LIN {X 0,Y 207.025,Z 158.787,A -85,B 0,C 180,E1 -21118.588,E2 -21118.588} C_VEL
LIN {X 0,Y 213.281,Z 171.917,A -85,B 0,C 180,E1 -21120.162,E2 -21120.162} C_VEL
LIN {X 0,Y 219.22,Z 186.796,A -85,B 0,C 180,E1 -21121.599,E2 -21121.599} C_VEL
LIN {X 0,Y 220.481,Z 191.391,A -85,B 0,C 180,E1 -21121.944,E2 -21121.944} C_VEL
LIN {X 0,Y 221.304,Z 196.769,A -85,B 0,C 180,E1 -21122.252,E2 -21122.252} C_VEL
LIN {X 0,Y 219.851,Z 234.463,A -85,B 0,C 180,E1 -21123.468,E2 -21123.468} C_VEL
LIN {X 0,Y 219.142,Z 244.352,A -85,B 0,C 180,E1 -21124.024,E2 -21124.024} C_VEL
LIN {X 0,Y 218.068,Z 254.849,A -85,B 0,C 180,E1 -21124.912,E2 -21124.912} C_VEL
LIN {X 0,Y 216.311,Z 266.211,A -85,B 0,C 180,E1 -21126.292,E2 -21126.292} C_VEL
LIN {X 0,Y 214.803,Z 274.591,A -85,B 0,C 180,E1 -21127.644,E2 -21127.644} C_VEL
LIN {X 0,Y 213.065,Z 282.507,A -85,B 0,C 180,E1 -21129.231,E2 -21129.231} C_VEL
LIN {X 0,Y 211.348,Z 289.887,A -85,B 0,C 180,E1 -21131.081,E2 -21131.081} C_VEL
LIN {X 0,Y 209.44,Z 297.362,A -85,B 0,C 180,E1 -21133.427,E2 -21133.427} C_VEL
LIN {X 0,Y 207.589,Z 304.212,A -85,B 0,C 180,E1 -21136.291,E2 -21136.291} C_VEL
LIN {X 0,Y 206.206,Z 309.389,A -85,B 0,C 180,E1 -21139.195,E2 -21139.195} C_VEL
LIN {X 0,Y 205.508,Z 312.044,A -85,B 0,C 180,E1 -21141.147,E2 -21141.147} C_VEL
LIN {X 0,Y 204.74,Z 315.32,A -85,B 0,C 180,E1 -21144.544,E2 -21144.544} C_VEL
LIN {X 0,Y 204.386,Z 317.015,A -85,B 0,C 180,E1 -21148.029,E2 -21148.029} C_VEL
LIN {X 0,Y 204.39,Z 317.318,A -85,B 0,C 180,E1 -21150,E2 -21150} C_VEL
LIN {X 0,Y 204.385,Z 317.039,A -85,B 0,C 180,E1 -21151.97,E2 -21151.97} C_VEL
LIN {X 0,Y 204.716,Z 315.5,A -85,B 0,C 180,E1 -21155.384,E2 -21155.384} C_VEL
LIN {X 0,Y 205.209,Z 313.362,A -85,B 0,C 180,E1 -21157.873,E2 -21157.873} C_VEL
LIN {X 0,Y 206.179,Z 309.614,A -85,B 0,C 180,E1 -21160.805,E2 -21160.805} C_VEL
LIN {X 0,Y 207.558,Z 304.498,A -85,B 0,C 180,E1 -21163.71,E2 -21163.71} C_VEL
LIN {X 0,Y 209.032,Z 298.993,A -85,B 0,C 180,E1 -21166.103,E2 -21166.103} C_VEL
LIN {X 0,Y 210.882,Z 292.07,A -85,B 0,C 180,E1 -21168.457,E2 -21168.457} C_VEL
LIN {X 0,Y 212.763,Z 284.122,A -85,B 0,C 180,E1 -21170.546,E2 -21170.546} C_VEL
LIN {X 0,Y 214.475,Z 276.541,A -85,B 0,C 180,E1 -21172.137,E2 -21172.137} C_VEL
LIN {X 0,Y 216.015,Z 268.593,A -85,B 0,C 180,E1 -21173.487,E2 -21173.487} C_VEL
LIN {X 0,Y 217.416,Z 260.376,A -85,B 0,C 180,E1 -21174.593,E2 -21174.593} C_VEL
LIN {X 0,Y 218.618,Z 251.281,A -85,B 0,C 180,E1 -21175.545,E2 -21175.545} C_VEL
LIN {X 0,Y 219.566,Z 240.802,A -85,B 0,C 180,E1 -21176.344,E2 -21176.344} C_VEL
LIN {X 0,Y 220.274,Z 226.937,A -85,B 0,C 180,E1 -21176.954,E2 -21176.954} C_VEL
LIN {X 0,Y 221.254,Z 195.857,A -85,B 0,C 180,E1 -21177.938,E2 -21177.938} C_VEL
LIN {X 0,Y 219.854,Z 188.323,A -85,B 0,C 180,E1 -21178.407,E2 -21178.407} C_VEL
LIN {X 0,Y 213.607,Z 172.604,A -85,B 0,C 180,E1 -21179.917,E2 -21179.917} C_VEL
LIN {X 0,Y 208.077,Z 161.104,A -85,B 0,C 180,E1 -21181.255,E2 -21181.255} C_VEL
LIN {X 0,Y 206.898,Z 158.307,A -85,B 0,C 180,E1 -21181.691,E2 -21181.691} C_VEL
LIN {X 0,Y 206.732,Z 157.678,A -85,B 0,C 180,E1 -21182.04,E2 -21182.04} C_VEL
LIN {X 0,Y 206.722,Z 157.517,A -85,B 0,C 180,E1 -21185.32,E2 -21185.32} C_VEL
LIN {X 0,Y 206.665,Z 157.531,A -85,B 0,C 180,E1 -21190.25,E2 -21190.25} C_VEL
LIN {X 0,Y 206.631,Z 157.549,A -85,B 0,C 180,E1 -21195.582,E2 -21195.582} C_VEL
LIN {X 0,Y 206.66,Z 157.542,A -85,B 0,C 180,E1 -21199.748,E2 -21199.748} C_VEL
LIN {X 0,Y 206.698,Z 157.542,A -85,B 0,C 180,E1 -21204.688,E2 -21204.688} C_VEL
LIN {X 0,Y 206.723,Z 157.548,A -85,B 0,C 180,E1 -21209.339,E2 -21209.339} C_VEL
LIN {X 0,Y 206.731,Z 157.525,A -85,B 0,C 180,E1 -21213.772,E2 -21213.772} C_VEL
LIN {X 0,Y 206.757,Z 157.542,A -85,B 0,C 180,E1 -21218.043,E2 -21218.043} C_VEL
LIN {X 0,Y 206.872,Z 157.503,A -85,B 0,C 180,E1 -21222.196,E2 -21222.196} C_VEL
LIN {X 0,Y 206.914,Z 157.523,A -85,B 0,C 180,E1 -21226.245,E2 -21226.245} C_VEL
LIN {X 0,Y 207.105,Z 157.474,A -85,B 0,C 180,E1 -21230.231,E2 -21230.231} C_VEL
LIN {X 0,Y 207.167,Z 157.468,A -85,B 0,C 180,E1 -21232.201,E2 -21232.201} C_VEL
LIN {X 0,Y 207.382,Z 157.456,A -85,B 0,C 180,E1 -21238.058,E2 -21238.058} C_VEL
LIN {X 0,Y 207.514,Z 157.421,A -85,B 0,C 180,E1 -21240,E2 -21240} C_VEL
LIN {X 0,Y 207.382,Z 157.44,A -85,B 0,C 180,E1 -21241.942,E2 -21241.942} C_VEL
LIN {X 0,Y 207.178,Z 157.481,A -85,B 0,C 180,E1 -21247.798,E2 -21247.798} C_VEL
LIN {X 0,Y 206.98,Z 157.493,A -85,B 0,C 180,E1 -21251.755,E2 -21251.755} C_VEL
LIN {X 0,Y 206.866,Z 157.528,A -85,B 0,C 180,E1 -21255.771,E2 -21255.771} C_VEL
LIN {X 0,Y 206.782,Z 157.516,A -85,B 0,C 180,E1 -21259.869,E2 -21259.869} C_VEL
LIN {X 0,Y 206.762,Z 157.542,A -85,B 0,C 180,E1 -21264.072,E2 -21264.072} C_VEL
LIN {X 0,Y 206.743,Z 157.526,A -85,B 0,C 180,E1 -21268.419,E2 -21268.419} C_VEL
LIN {X 0,Y 206.701,Z 157.544,A -85,B 0,C 180,E1 -21272.957,E2 -21272.957} C_VEL
LIN {X 0,Y 206.679,Z 157.553,A -85,B 0,C 180,E1 -21277.74,E2 -21277.74} C_VEL
LIN {X 0,Y 206.639,Z 157.518,A -85,B 0,C 180,E1 -21281.562,E2 -21281.562} C_VEL
LIN {X 0,Y 206.629,Z 157.526,A -85,B 0,C 180,E1 -21285.583,E2 -21285.583} C_VEL
LIN {X 0,Y 206.658,Z 157.54,A -85,B 0,C 180,E1 -21289.749,E2 -21289.749} C_VEL
LIN {X 0,Y 206.714,Z 157.652,A -85,B 0,C 180,E1 -21294.558,E2 -21294.558} C_VEL
LIN {X 0,Y 208.276,Z 164.486,A -85,B 0,C 180,E1 -21298.581,E2 -21298.581} C_VEL
LIN {X 0,Y 209.79,Z 168.116,A -85,B 0,C 180,E1 -21299.094,E2 -21299.094} C_VEL
LIN {X 0,Y 213.712,Z 177.001,A -85,B 0,C 180,E1 -21300.057,E2 -21300.057} C_VEL
LIN {X 0,Y 214.926,Z 182.58,A -85,B 0,C 180,E1 -21300.452,E2 -21300.452} C_VEL
LIN {X 0,Y 215.138,Z 188.446,A -85,B 0,C 180,E1 -21300.704,E2 -21300.704} C_VEL
LIN {X 0,Y 214.129,Z 204.462,A -85,B 0,C 180,E1 -21301.155,E2 -21301.155} C_VEL
LIN {X 0,Y 214.248,Z 208.452,A -85,B 0,C 180,E1 -21301.322,E2 -21301.322} C_VEL
LIN {X 0,Y 214.544,Z 211.919,A -85,B 0,C 180,E1 -21301.494,E2 -21301.494} C_VEL
LIN {X 0,Y 213.364,Z 242.504,A -85,B 0,C 180,E1 -21302.539,E2 -21302.539} C_VEL
LIN {X 0,Y 212.457,Z 252.749,A -85,B 0,C 180,E1 -21303.145,E2 -21303.145} C_VEL
LIN {X 0,Y 211.077,Z 263.496,A -85,B 0,C 180,E1 -21304.114,E2 -21304.114} C_VEL
LIN {X 0,Y 209.3,Z 273.86,A -85,B 0,C 180,E1 -21305.448,E2 -21305.448} C_VEL
LIN {X 0,Y 207.628,Z 282.146,A -85,B 0,C 180,E1 -21306.828,E2 -21306.828} C_VEL
LIN {X 0,Y 205.824,Z 289.992,A -85,B 0,C 180,E1 -21308.466,E2 -21308.466} C_VEL
LIN {X 0,Y 203.943,Z 297.33,A -85,B 0,C 180,E1 -21310.368,E2 -21310.368} C_VEL
LIN {X 0,Y 201.943,Z 304.775,A -85,B 0,C 180,E1 -21312.794,E2 -21312.794} C_VEL
LIN {X 0,Y 200.353,Z 310.611,A -85,B 0,C 180,E1 -21315.267,E2 -21315.267} C_VEL
LIN {X 0,Y 199.065,Z 315.214,A -85,B 0,C 180,E1 -21317.771,E2 -21317.771} C_VEL
LIN {X 0,Y 198.362,Z 318.207,A -85,B 0,C 180,E1 -21319.797,E2 -21319.797} C_VEL
LIN {X 0,Y 197.78,Z 320.53,A -85,B 0,C 180,E1 -21321.829,E2 -21321.829} C_VEL
LIN {X 0,Y 197.427,Z 322.272,A -85,B 0,C 180,E1 -21323.87,E2 -21323.87} C_VEL
LIN {X 0,Y 197.237,Z 323.613,A -85,B 0,C 180,E1 -21326.113,E2 -21326.113} C_VEL
LIN {X 0,Y 197.214,Z 324.293,A -85,B 0,C 180,E1 -21327.958,E2 -21327.958} C_VEL
LIN {X 0,Y 197.252,Z 324.585,A -85,B 0,C 180,E1 -21330,E2 -21330} C_VEL
LIN {X 0,Y 197.214,Z 324.283,A -85,B 0,C 180,E1 -21332.043,E2 -21332.043} C_VEL
LIN {X 0,Y 197.25,Z 323.49,A -85,B 0,C 180,E1 -21334.087,E2 -21334.087} C_VEL
LIN {X 0,Y 197.43,Z 322.223,A -85,B 0,C 180,E1 -21336.131,E2 -21336.131} C_VEL
LIN {X 0,Y 198.004,Z 319.305,A -85,B 0,C 180,E1 -21339.191,E2 -21339.191} C_VEL
LIN {X 0,Y 198.649,Z 316.646,A -85,B 0,C 180,E1 -21341.221,E2 -21341.221} C_VEL
LIN {X 0,Y 200.061,Z 311.454,A -85,B 0,C 180,E1 -21344.236,E2 -21344.236} C_VEL
LIN {X 0,Y 201.922,Z 304.606,A -85,B 0,C 180,E1 -21347.209,E2 -21347.209} C_VEL
LIN {X 0,Y 203.932,Z 297.128,A -85,B 0,C 180,E1 -21349.634,E2 -21349.634} C_VEL
LIN {X 0,Y 205.828,Z 289.754,A -85,B 0,C 180,E1 -21351.535,E2 -21351.535} C_VEL
LIN {X 0,Y 207.584,Z 281.852,A -85,B 0,C 180,E1 -21353.178,E2 -21353.178} C_VEL
LIN {X 0,Y 209.567,Z 272.214,A -85,B 0,C 180,E1 -21354.746,E2 -21354.746} C_VEL
LIN {X 0,Y 211.277,Z 261.067,A -85,B 0,C 180,E1 -21356.086,E2 -21356.086} C_VEL
LIN {X 0,Y 212.53,Z 251.125,A -85,B 0,C 180,E1 -21356.912,E2 -21356.912} C_VEL
LIN {X 0,Y 213.384,Z 241.25,A -85,B 0,C 180,E1 -21357.459,E2 -21357.459} C_VEL
LIN {X 0,Y 214.439,Z 210.557,A -85,B 0,C 180,E1 -21358.508,E2 -21358.508} C_VEL
LIN {X 0,Y 211.33,Z 188.673,A -85,B 0,C 180,E1 -21359.799,E2 -21359.799} C_VEL
LIN {X 0,Y 205.481,Z 174.284,A -85,B 0,C 180,E1 -21361.306,E2 -21361.306} C_VEL
LIN {X 0,Y 201.105,Z 164.731,A -85,B 0,C 180,E1 -21362.512,E2 -21362.512} C_VEL
LIN {X 0,Y 200.705,Z 163.01,A -85,B 0,C 180,E1 -21363.337,E2 -21363.337} C_VEL
LIN {X 0,Y 199.673,Z 158.489,A -85,B 0,C 180,E1 -21366.258,E2 -21366.258} C_VEL
LIN {X 0,Y 199.608,Z 158.407,A -85,B 0,C 180,E1 -21369.329,E2 -21369.329} C_VEL
LIN {X 0,Y 199.573,Z 158.437,A -85,B 0,C 180,E1 -21372.31,E2 -21372.31} C_VEL
LIN {X 0,Y 199.577,Z 158.389,A -85,B 0,C 180,E1 -21375.228,E2 -21375.228} C_VEL
LIN {X 0,Y 199.578,Z 158.39,A -85,B 0,C 180,E1 -21378.005,E2 -21378.005} C_VEL
LIN {X 0,Y 199.612,Z 158.43,A -85,B 0,C 180,E1 -21380.768,E2 -21380.768} C_VEL
LIN {X 0,Y 199.614,Z 158.418,A -85,B 0,C 180,E1 -21385.714,E2 -21385.714} C_VEL
LIN {X 0,Y 199.702,Z 158.422,A -85,B 0,C 180,E1 -21388.138,E2 -21388.138} C_VEL
LIN {X 0,Y 199.688,Z 158.402,A -85,B 0,C 180,E1 -21392.772,E2 -21392.772} C_VEL
LIN {X 0,Y 199.74,Z 158.414,A -85,B 0,C 180,E1 -21397.23,E2 -21397.23} C_VEL
LIN {X 0,Y 199.799,Z 158.392,A -85,B 0,C 180,E1 -21401.758,E2 -21401.758} C_VEL
LIN {X 0,Y 199.838,Z 158.403,A -85,B 0,C 180,E1 -21405.749,E2 -21405.749} C_VEL
LIN {X 0,Y 200.024,Z 158.352,A -85,B 0,C 180,E1 -21409.882,E2 -21409.882} C_VEL
LIN {X 0,Y 200.029,Z 158.38,A -85,B 0,C 180,E1 -21413.95,E2 -21413.95} C_VEL
LIN {X 0,Y 200.323,Z 158.318,A -85,B 0,C 180,E1 -21417.99,E2 -21417.99} C_VEL
LIN {X 0,Y 200.479,Z 158.296,A -85,B 0,C 180,E1 -21420,E2 -21420} C_VEL
LIN {X 0,Y 200.034,Z 158.382,A -85,B 0,C 180,E1 -21424.03,E2 -21424.03} C_VEL
LIN {X 0,Y 200.114,Z 158.343,A -85,B 0,C 180,E1 -21428.076,E2 -21428.076} C_VEL
LIN {X 0,Y 199.917,Z 158.39,A -85,B 0,C 180,E1 -21432.177,E2 -21432.177} C_VEL
LIN {X 0,Y 199.807,Z 158.395,A -85,B 0,C 180,E1 -21436.343,E2 -21436.343} C_VEL
LIN {X 0,Y 199.703,Z 158.413,A -85,B 0,C 180,E1 -21440.605,E2 -21440.605} C_VEL
LIN {X 0,Y 199.675,Z 158.411,A -85,B 0,C 180,E1 -21444.984,E2 -21444.984} C_VEL
LIN {X 0,Y 199.677,Z 158.424,A -85,B 0,C 180,E1 -21449.522,E2 -21449.522} C_VEL
LIN {X 0,Y 199.68,Z 158.414,A -85,B 0,C 180,E1 -21452.358,E2 -21452.358} C_VEL
LIN {X 0,Y 199.625,Z 158.432,A -85,B 0,C 180,E1 -21456.763,E2 -21456.763} C_VEL
LIN {X 0,Y 199.61,Z 158.422,A -85,B 0,C 180,E1 -21459.328,E2 -21459.328} C_VEL
LIN {X 0,Y 199.576,Z 158.438,A -85,B 0,C 180,E1 -21462.31,E2 -21462.31} C_VEL
LIN {X 0,Y 199.579,Z 158.413,A -85,B 0,C 180,E1 -21465.228,E2 -21465.228} C_VEL
LIN {X 0,Y 199.641,Z 158.419,A -85,B 0,C 180,E1 -21470.679,E2 -21470.679} C_VEL
LIN {X 0,Y 199.636,Z 158.399,A -85,B 0,C 180,E1 -21475.718,E2 -21475.718} C_VEL
LIN {X 0,Y 199.714,Z 158.737,A -85,B 0,C 180,E1 -21477.093,E2 -21477.093} C_VEL
LIN {X 0,Y 200.101,Z 160.119,A -85,B 0,C 180,E1 -21477.452,E2 -21477.452} C_VEL
LIN {X 0,Y 203.509,Z 166.286,A -85,B 0,C 180,E1 -21478.333,E2 -21478.333} C_VEL
LIN {X 0,Y 210.222,Z 181.264,A -85,B 0,C 180,E1 -21480.042,E2 -21480.042} C_VEL
LIN {X 0,Y 214.246,Z 192.387,A -85,B 0,C 180,E1 -21481.083,E2 -21481.083} C_VEL
LIN {X 0,Y 215.01,Z 197.207,A -85,B 0,C 180,E1 -21481.376,E2 -21481.376} C_VEL
LIN {X 0,Y 213.523,Z 234.798,A -85,B 0,C 180,E1 -21482.626,E2 -21482.626} C_VEL
LIN {X 0,Y 212.788,Z 244.531,A -85,B 0,C 180,E1 -21483.19,E2 -21483.19} C_VEL
LIN {X 0,Y 211.656,Z 255.205,A -85,B 0,C 180,E1 -21484.121,E2 -21484.121} C_VEL
LIN {X 0,Y 209.848,Z 266.344,A -85,B 0,C 180,E1 -21485.515,E2 -21485.515} C_VEL
LIN {X 0,Y 208.27,Z 274.723,A -85,B 0,C 180,E1 -21486.903,E2 -21486.903} C_VEL
LIN {X 0,Y 206.459,Z 282.638,A -85,B 0,C 180,E1 -21488.534,E2 -21488.534} C_VEL
LIN {X 0,Y 205.046,Z 288.32,A -85,B 0,C 180,E1 -21489.955,E2 -21489.955} C_VEL
LIN {X 0,Y 203.393,Z 294.666,A -85,B 0,C 180,E1 -21491.881,E2 -21491.881} C_VEL
LIN {X 0,Y 201.929,Z 299.94,A -85,B 0,C 180,E1 -21493.833,E2 -21493.833} C_VEL
LIN {X 0,Y 200.693,Z 304.342,A -85,B 0,C 180,E1 -21495.81,E2 -21495.81} C_VEL
LIN {X 0,Y 199.23,Z 309.519,A -85,B 0,C 180,E1 -21498.812,E2 -21498.812} C_VEL
LIN {X 0,Y 198.486,Z 312.173,A -85,B 0,C 180,E1 -21500.831,E2 -21500.831} C_VEL
LIN {X 0,Y 197.767,Z 315.079,A -85,B 0,C 180,E1 -21503.88,E2 -21503.88} C_VEL
LIN {X 0,Y 197.467,Z 316.345,A -85,B 0,C 180,E1 -21505.918,E2 -21505.918} C_VEL
LIN {X 0,Y 197.299,Z 317.143,A -85,B 0,C 180,E1 -21507.958,E2 -21507.958} C_VEL
LIN {X 0,Y 197.296,Z 317.446,A -85,B 0,C 180,E1 -21510,E2 -21510} C_VEL
LIN {X 0,Y 197.298,Z 317.167,A -85,B 0,C 180,E1 -21512.041,E2 -21512.041} C_VEL
LIN {X 0,Y 197.6,Z 315.877,A -85,B 0,C 180,E1 -21515.205,E2 -21515.205} C_VEL
LIN {X 0,Y 198.175,Z 313.49,A -85,B 0,C 180,E1 -21518.155,E2 -21518.155} C_VEL
LIN {X 0,Y 199.204,Z 309.741,A -85,B 0,C 180,E1 -21521.188,E2 -21521.188} C_VEL
LIN {X 0,Y 200.657,Z 304.625,A -85,B 0,C 180,E1 -21524.192,E2 -21524.192} C_VEL
LIN {X 0,Y 202.219,Z 299.119,A -85,B 0,C 180,E1 -21526.661,E2 -21526.661} C_VEL
LIN {X 0,Y 204.159,Z 292.196,A -85,B 0,C 180,E1 -21529.088,E2 -21529.088} C_VEL
LIN {X 0,Y 206.148,Z 284.247,A -85,B 0,C 180,E1 -21531.237,E2 -21531.237} C_VEL
LIN {X 0,Y 207.937,Z 276.665,A -85,B 0,C 180,E1 -21532.872,E2 -21532.872} C_VEL
LIN {X 0,Y 209.542,Z 268.716,A -85,B 0,C 180,E1 -21534.258,E2 -21534.258} C_VEL
LIN {X 0,Y 210.987,Z 260.498,A -85,B 0,C 180,E1 -21535.395,E2 -21535.395} C_VEL
LIN {X 0,Y 212.159,Z 252.232,A -85,B 0,C 180,E1 -21536.291,E2 -21536.291} C_VEL
LIN {X 0,Y 213.083,Z 242.81,A -85,B 0,C 180,E1 -21537.06,E2 -21537.06} C_VEL
LIN {X 0,Y 213.691,Z 233.428,A -85,B 0,C 180,E1 -21537.574,E2 -21537.574} C_VEL
LIN {X 0,Y 215.027,Z 197.05,A -85,B 0,C 180,E1 -21538.781,E2 -21538.781} C_VEL
LIN {X 0,Y 213.929,Z 191.058,A -85,B 0,C 180,E1 -21539.169,E2 -21539.169} C_VEL
LIN {X 0,Y 208.339,Z 176.751,A -85,B 0,C 180,E1 -21540.595,E2 -21540.595} C_VEL
LIN {X 0,Y 202.889,Z 165.209,A -85,B 0,C 180,E1 -21541.984,E2 -21541.984} C_VEL
LIN {X 0,Y 200.65,Z 161.212,A -85,B 0,C 180,E1 -21542.552,E2 -21542.552} C_VEL
LIN {X 0,Y 199.794,Z 159.117,A -85,B 0,C 180,E1 -21542.912,E2 -21542.912} C_VEL
LIN {X 0,Y 199.67,Z 158.533,A -85,B 0,C 180,E1 -21543.244,E2 -21543.244} C_VEL
LIN {X 0,Y 199.619,Z 158.41,A -85,B 0,C 180,E1 -21546.763,E2 -21546.763} C_VEL
LIN {X 0,Y 199.639,Z 158.424,A -85,B 0,C 180,E1 -21549.32,E2 -21549.32} C_VEL
LIN {X 0,Y 199.577,Z 158.409,A -85,B 0,C 180,E1 -21554.771,E2 -21554.771} C_VEL
LIN {X 0,Y 199.578,Z 158.437,A -85,B 0,C 180,E1 -21558.004,E2 -21558.004} C_VEL
LIN {X 0,Y 199.61,Z 158.421,A -85,B 0,C 180,E1 -21560.767,E2 -21560.767} C_VEL
LIN {X 0,Y 199.612,Z 158.415,A -85,B 0,C 180,E1 -21565.713,E2 -21565.713} C_VEL
LIN {X 0,Y 199.7,Z 158.416,A -85,B 0,C 180,E1 -21568.137,E2 -21568.137} C_VEL
LIN {X 0,Y 199.686,Z 158.404,A -85,B 0,C 180,E1 -21572.771,E2 -21572.771} C_VEL
LIN {X 0,Y 199.738,Z 158.417,A -85,B 0,C 180,E1 -21577.229,E2 -21577.229} C_VEL
LIN {X 0,Y 199.796,Z 158.383,A -85,B 0,C 180,E1 -21581.757,E2 -21581.757} C_VEL
LIN {X 0,Y 199.848,Z 158.402,A -85,B 0,C 180,E1 -21585.749,E2 -21585.749} C_VEL
LIN {X 0,Y 200.069,Z 158.352,A -85,B 0,C 180,E1 -21589.884,E2 -21589.884} C_VEL
LIN {X 0,Y 200.035,Z 158.372,A -85,B 0,C 180,E1 -21593.949,E2 -21593.949} C_VEL
LIN {X 0,Y 200.322,Z 158.335,A -85,B 0,C 180,E1 -21597.989,E2 -21597.989} C_VEL
LIN {X 0,Y 200.479,Z 158.297,A -85,B 0,C 180,E1 -21600,E2 -21600} C_VEL
LIN {X 0,Y 200.031,Z 158.374,A -85,B 0,C 180,E1 -21604.029,E2 -21604.029} C_VEL
LIN {X 0,Y 200.119,Z 158.359,A -85,B 0,C 180,E1 -21608.075,E2 -21608.075} C_VEL
LIN {X 0,Y 199.913,Z 158.377,A -85,B 0,C 180,E1 -21612.177,E2 -21612.177} C_VEL
LIN {X 0,Y 199.804,Z 158.406,A -85,B 0,C 180,E1 -21616.343,E2 -21616.343} C_VEL
LIN {X 0,Y 199.699,Z 158.401,A -85,B 0,C 180,E1 -21620.605,E2 -21620.605} C_VEL
LIN {X 0,Y 199.672,Z 158.422,A -85,B 0,C 180,E1 -21624.984,E2 -21624.984} C_VEL
LIN {X 0,Y 199.673,Z 158.415,A -85,B 0,C 180,E1 -21629.522,E2 -21629.522} C_VEL
LIN {X 0,Y 199.676,Z 158.423,A -85,B 0,C 180,E1 -21632.358,E2 -21632.358} C_VEL
LIN {X 0,Y 199.622,Z 158.428,A -85,B 0,C 180,E1 -21636.763,E2 -21636.763} C_VEL
LIN {X 0,Y 199.607,Z 158.428,A -85,B 0,C 180,E1 -21639.328,E2 -21639.328} C_VEL
LIN {X 0,Y 199.57,Z 158.388,A -85,B 0,C 180,E1 -21642.31,E2 -21642.31} C_VEL
LIN {X 0,Y 199.575,Z 158.396,A -85,B 0,C 180,E1 -21645.228,E2 -21645.228} C_VEL
LIN {X 0,Y 199.577,Z 158.439,A -85,B 0,C 180,E1 -21648.005,E2 -21648.005} C_VEL
LIN {X 0,Y 199.653,Z 158.405,A -85,B 0,C 180,E1 -21653.244,E2 -21653.244} C_VEL
LIN {X 0,Y 199.727,Z 158.927,A -85,B 0,C 180,E1 -21654.03,E2 -21654.03} C_VEL
LIN {X 0,Y 201.015,Z 164.444,A -85,B 0,C 180,E1 -21657.335,E2 -21657.335} C_VEL
LIN {X 0,Y 203.312,Z 169.666,A -85,B 0,C 180,E1 -21658.063,E2 -21658.063} C_VEL
LIN {X 0,Y 208.434,Z 181.104,A -85,B 0,C 180,E1 -21659.382,E2 -21659.382} C_VEL
LIN {X 0,Y 211.571,Z 189.597,A -85,B 0,C 180,E1 -21660.207,E2 -21660.207} C_VEL
LIN {X 0,Y 214.248,Z 208.452,A -85,B 0,C 180,E1 -21661.322,E2 -21661.322} C_VEL
LIN {X 0,Y 214.19,Z 212.339,A -85,B 0,C 180,E1 -21661.454,E2 -21661.454} C_VEL
LIN {X 0,Y 213.558,Z 216.217,A -85,B 0,C 180,E1 -21661.496,E2 -21661.496} C_VEL
LIN {X 0,Y 208.229,Z 233.389,A -85,B 0,C 180,E1 -21661.352,E2 -21661.352} C_VEL
LIN {X 0,Y 207.287,Z 239.256,A -85,B 0,C 180,E1 -21661.496,E2 -21661.496} C_VEL
LIN {X 0,Y 206.51,Z 249.311,A -85,B 0,C 180,E1 -21662.031,E2 -21662.031} C_VEL
LIN {X 0,Y 205.36,Z 258.749,A -85,B 0,C 180,E1 -21662.788,E2 -21662.788} C_VEL
LIN {X 0,Y 203.979,Z 267.807,A -85,B 0,C 180,E1 -21663.794,E2 -21663.794} C_VEL
LIN {X 0,Y 202.24,Z 276.884,A -85,B 0,C 180,E1 -21665.107,E2 -21665.107} C_VEL
LIN {X 0,Y 200.02,Z 286.799,A -85,B 0,C 180,E1 -21666.991,E2 -21666.991} C_VEL
LIN {X 0,Y 197.726,Z 295.497,A -85,B 0,C 180,E1 -21669.18,E2 -21669.18} C_VEL
LIN {X 0,Y 195.949,Z 301.815,A -85,B 0,C 180,E1 -21671.168,E2 -21671.168} C_VEL
LIN {X 0,Y 194.402,Z 307.064,A -85,B 0,C 180,E1 -21673.19,E2 -21673.19} C_VEL
LIN {X 0,Y 193.175,Z 311.443,A -85,B 0,C 180,E1 -21675.246,E2 -21675.246} C_VEL
LIN {X 0,Y 191.716,Z 316.609,A -85,B 0,C 180,E1 -21678.369,E2 -21678.369} C_VEL
LIN {X 0,Y 190.748,Z 320.403,A -85,B 0,C 180,E1 -21681.526,E2 -21681.526} C_VEL
LIN {X 0,Y 190.369,Z 322.144,A -85,B 0,C 180,E1 -21683.642,E2 -21683.642} C_VEL
LIN {X 0,Y 190.142,Z 323.657,A -85,B 0,C 180,E1 -21686.344,E2 -21686.344} C_VEL
LIN {X 0,Y 190.161,Z 324.457,A -85,B 0,C 180,E1 -21690.001,E2 -21690.001} C_VEL
LIN {X 0,Y 190.142,Z 323.627,A -85,B 0,C 180,E1 -21693.657,E2 -21693.657} C_VEL
LIN {X 0,Y 190.372,Z 322.094,A -85,B 0,C 180,E1 -21696.359,E2 -21696.359} C_VEL
LIN {X 0,Y 190.998,Z 319.176,A -85,B 0,C 180,E1 -21699.532,E2 -21699.532} C_VEL
LIN {X 0,Y 191.685,Z 316.516,A -85,B 0,C 180,E1 -21701.634,E2 -21701.634} C_VEL
LIN {X 0,Y 193.172,Z 311.323,A -85,B 0,C 180,E1 -21704.755,E2 -21704.755} C_VEL
LIN {X 0,Y 195.145,Z 304.475,A -85,B 0,C 180,E1 -21707.826,E2 -21707.826} C_VEL
LIN {X 0,Y 197.251,Z 296.997,A -85,B 0,C 180,E1 -21710.328,E2 -21710.328} C_VEL
LIN {X 0,Y 199.232,Z 289.622,A -85,B 0,C 180,E1 -21712.285,E2 -21712.285} C_VEL
LIN {X 0,Y 201.076,Z 281.72,A -85,B 0,C 180,E1 -21713.974,E2 -21713.974} C_VEL
LIN {X 0,Y 203.062,Z 272.531,A -85,B 0,C 180,E1 -21715.513,E2 -21715.513} C_VEL
LIN {X 0,Y 204.763,Z 262.276,A -85,B 0,C 180,E1 -21716.825,E2 -21716.825} C_VEL
LIN {X 0,Y 206.229,Z 250.986,A -85,B 0,C 180,E1 -21717.804,E2 -21717.804} C_VEL
LIN {X 0,Y 207.114,Z 241.105,A -85,B 0,C 180,E1 -21718.364,E2 -21718.364} C_VEL
LIN {X 0,Y 208.201,Z 211.301,A -85,B 0,C 180,E1 -21719.41,E2 -21719.41} C_VEL
LIN {X 0,Y 205.304,Z 190.857,A -85,B 0,C 180,E1 -21720.674,E2 -21720.674} C_VEL
LIN {X 0,Y 199.891,Z 177.49,A -85,B 0,C 180,E1 -21722.146,E2 -21722.146} C_VEL
LIN {X 0,Y 193.873,Z 164.661,A -85,B 0,C 180,E1 -21723.873,E2 -21723.873} C_VEL
LIN {X 0,Y 193.55,Z 163.504,A -85,B 0,C 180,E1 -21724.374,E2 -21724.374} C_VEL
LIN {X 0,Y 192.605,Z 159.381,A -85,B 0,C 180,E1 -21727.149,E2 -21727.149} C_VEL
LIN {X 0,Y 192.513,Z 159.313,A -85,B 0,C 180,E1 -21731.081,E2 -21731.081} C_VEL
LIN {X 0,Y 192.489,Z 159.264,A -85,B 0,C 180,E1 -21736.076,E2 -21736.076} C_VEL
LIN {X 0,Y 192.519,Z 159.303,A -85,B 0,C 180,E1 -21740.052,E2 -21740.052} C_VEL
LIN {X 0,Y 192.562,Z 159.297,A -85,B 0,C 180,E1 -21744.271,E2 -21744.271} C_VEL
LIN {X 0,Y 192.612,Z 159.299,A -85,B 0,C 180,E1 -21747.059,E2 -21747.059} C_VEL
LIN {X 0,Y 192.666,Z 159.276,A -85,B 0,C 180,E1 -21751.692,E2 -21751.692} C_VEL
LIN {X 0,Y 192.708,Z 159.293,A -85,B 0,C 180,E1 -21756.349,E2 -21756.349} C_VEL
LIN {X 0,Y 192.734,Z 159.268,A -85,B 0,C 180,E1 -21761.458,E2 -21761.458} C_VEL
LIN {X 0,Y 192.766,Z 159.285,A -85,B 0,C 180,E1 -21765.214,E2 -21765.214} C_VEL
LIN {X 0,Y 192.947,Z 159.232,A -85,B 0,C 180,E1 -21769.567,E2 -21769.567} C_VEL
LIN {X 0,Y 193.044,Z 159.236,A -85,B 0,C 180,E1 -21771.627,E2 -21771.627} C_VEL
LIN {X 0,Y 193.265,Z 159.197,A -85,B 0,C 180,E1 -21777.916,E2 -21777.916} C_VEL
LIN {X 0,Y 193.443,Z 159.171,A -85,B 0,C 180,E1 -21780,E2 -21780} C_VEL
LIN {X 0,Y 192.98,Z 159.259,A -85,B 0,C 180,E1 -21784.177,E2 -21784.177} C_VEL
LIN {X 0,Y 193.065,Z 159.219,A -85,B 0,C 180,E1 -21788.373,E2 -21788.373} C_VEL
LIN {X 0,Y 192.856,Z 159.272,A -85,B 0,C 180,E1 -21792.63,E2 -21792.63} C_VEL
LIN {X 0,Y 192.76,Z 159.264,A -85,B 0,C 180,E1 -21796.959,E2 -21796.959} C_VEL
LIN {X 0,Y 192.639,Z 159.297,A -85,B 0,C 180,E1 -21801.397,E2 -21801.397} C_VEL
LIN {X 0,Y 192.667,Z 159.291,A -85,B 0,C 180,E1 -21804.225,E2 -21804.225} C_VEL
LIN {X 0,Y 192.652,Z 159.293,A -85,B 0,C 180,E1 -21808.892,E2 -21808.892} C_VEL
LIN {X 0,Y 192.601,Z 159.288,A -85,B 0,C 180,E1 -21813.186,E2 -21813.186} C_VEL
LIN {X 0,Y 192.553,Z 159.307,A -85,B 0,C 180,E1 -21818.352,E2 -21818.352} C_VEL
LIN {X 0,Y 192.513,Z 159.319,A -85,B 0,C 180,E1 -21823.102,E2 -21823.102} C_VEL
LIN {X 0,Y 192.492,Z 159.275,A -85,B 0,C 180,E1 -21826.905,E2 -21826.905} C_VEL
LIN {X 0,Y 192.57,Z 159.312,A -85,B 0,C 180,E1 -21831.652,E2 -21831.652} C_VEL
LIN {X 0,Y 192.634,Z 159.466,A -85,B 0,C 180,E1 -21835.652,E2 -21835.652} C_VEL
LIN {X 0,Y 192.845,Z 160.453,A -85,B 0,C 180,E1 -21836.058,E2 -21836.058} C_VEL
LIN {X 0,Y 198.456,Z 170.644,A -85,B 0,C 180,E1 -21837.607,E2 -21837.607} C_VEL
LIN {X 0,Y 204.768,Z 184.91,A -85,B 0,C 180,E1 -21839.299,E2 -21839.299} C_VEL
LIN {X 0,Y 208.232,Z 194.678,A -85,B 0,C 180,E1 -21840.249,E2 -21840.249} C_VEL
LIN {X 0,Y 208.808,Z 198.406,A -85,B 0,C 180,E1 -21840.484,E2 -21840.484} C_VEL
LIN {X 0,Y 207.242,Z 235.122,A -85,B 0,C 180,E1 -21841.733,E2 -21841.733} C_VEL
LIN {X 0,Y 206.455,Z 245.188,A -85,B 0,C 180,E1 -21842.341,E2 -21842.341} C_VEL
LIN {X 0,Y 205.12,Z 256.721,A -85,B 0,C 180,E1 -21843.411,E2 -21843.411} C_VEL
LIN {X 0,Y 203.428,Z 266.477,A -85,B 0,C 180,E1 -21844.689,E2 -21844.689} C_VEL
LIN {X 0,Y 201.778,Z 274.856,A -85,B 0,C 180,E1 -21846.114,E2 -21846.114} C_VEL
LIN {X 0,Y 199.877,Z 282.77,A -85,B 0,C 180,E1 -21847.791,E2 -21847.791} C_VEL
LIN {X 0,Y 198.404,Z 288.451,A -85,B 0,C 180,E1 -21849.253,E2 -21849.253} C_VEL
LIN {X 0,Y 196.655,Z 294.797,A -85,B 0,C 180,E1 -21851.237,E2 -21851.237} C_VEL
LIN {X 0,Y 195.126,Z 300.07,A -85,B 0,C 180,E1 -21853.253,E2 -21853.253} C_VEL
LIN {X 0,Y 193.8,Z 304.472,A -85,B 0,C 180,E1 -21855.294,E2 -21855.294} C_VEL
LIN {X 0,Y 192.277,Z 309.648,A -85,B 0,C 180,E1 -21858.402,E2 -21858.402} C_VEL
LIN {X 0,Y 191.486,Z 312.303,A -85,B 0,C 180,E1 -21860.493,E2 -21860.493} C_VEL
LIN {X 0,Y 190.725,Z 315.207,A -85,B 0,C 180,E1 -21863.653,E2 -21863.653} C_VEL
LIN {X 0,Y 190.405,Z 316.474,A -85,B 0,C 180,E1 -21865.766,E2 -21865.766} C_VEL
LIN {X 0,Y 190.214,Z 317.272,A -85,B 0,C 180,E1 -21867.882,E2 -21867.882} C_VEL
LIN {X 0,Y 190.204,Z 317.574,A -85,B 0,C 180,E1 -21869.999,E2 -21869.999} C_VEL
LIN {X 0,Y 190.213,Z 317.295,A -85,B 0,C 180,E1 -21872.117,E2 -21872.117} C_VEL
LIN {X 0,Y 190.497,Z 316.174,A -85,B 0,C 180,E1 -21875.052,E2 -21875.052} C_VEL
LIN {X 0,Y 191.14,Z 313.617,A -85,B 0,C 180,E1 -21878.457,E2 -21878.457} C_VEL
LIN {X 0,Y 192.249,Z 309.869,A -85,B 0,C 180,E1 -21881.598,E2 -21881.598} C_VEL
LIN {X 0,Y 193.764,Z 304.752,A -85,B 0,C 180,E1 -21884.708,E2 -21884.708} C_VEL
LIN {X 0,Y 195.437,Z 299.246,A -85,B 0,C 180,E1 -21887.257,E2 -21887.257} C_VEL
LIN {X 0,Y 197.468,Z 292.322,A -85,B 0,C 180,E1 -21889.761,E2 -21889.761} C_VEL
LIN {X 0,Y 199.566,Z 284.372,A -85,B 0,C 180,E1 -21891.973,E2 -21891.973} C_VEL
LIN {X 0,Y 201.434,Z 276.789,A -85,B 0,C 180,E1 -21893.655,E2 -21893.655} C_VEL
LIN {X 0,Y 203.108,Z 268.839,A -85,B 0,C 180,E1 -21895.079,E2 -21895.079} C_VEL
LIN {X 0,Y 204.593,Z 260.62,A -85,B 0,C 180,E1 -21896.248,E2 -21896.248} C_VEL
LIN {X 0,Y 205.748,Z 252.969,A -85,B 0,C 180,E1 -21897.106,E2 -21897.106} C_VEL
LIN {X 0,Y 206.766,Z 243.1,A -85,B 0,C 180,E1 -21897.943,E2 -21897.943} C_VEL
LIN {X 0,Y 207.4,Z 234.173,A -85,B 0,C 180,E1 -21898.451,E2 -21898.451} C_VEL
LIN {X 0,Y 208.819,Z 197.935,A -85,B 0,C 180,E1 -21899.691,E2 -21899.691} C_VEL
LIN {X 0,Y 207.896,Z 193.303,A -85,B 0,C 180,E1 -21900.018,E2 -21900.018} C_VEL
LIN {X 0,Y 202.477,Z 179.322,A -85,B 0,C 180,E1 -21901.48,E2 -21901.48} C_VEL
LIN {X 0,Y 196.569,Z 166.923,A -85,B 0,C 180,E1 -21903.073,E2 -21903.073} C_VEL
LIN {X 0,Y 193.827,Z 162.514,A -85,B 0,C 180,E1 -21903.797,E2 -21903.797} C_VEL
LIN {X 0,Y 192.726,Z 160.012,A -85,B 0,C 180,E1 -21904.234,E2 -21904.234} C_VEL
LIN {X 0,Y 192.6,Z 159.379,A -85,B 0,C 180,E1 -21904.625,E2 -21904.625} C_VEL
LIN {X 0,Y 192.568,Z 159.312,A -85,B 0,C 180,E1 -21908.347,E2 -21908.347} C_VEL
LIN {X 0,Y 192.489,Z 159.273,A -85,B 0,C 180,E1 -21913.095,E2 -21913.095} C_VEL
LIN {X 0,Y 192.511,Z 159.319,A -85,B 0,C 180,E1 -21916.897,E2 -21916.897} C_VEL
LIN {X 0,Y 192.551,Z 159.306,A -85,B 0,C 180,E1 -21921.648,E2 -21921.648} C_VEL
LIN {X 0,Y 192.598,Z 159.288,A -85,B 0,C 180,E1 -21926.814,E2 -21926.814} C_VEL
LIN {X 0,Y 192.664,Z 159.288,A -85,B 0,C 180,E1 -21931.692,E2 -21931.692} C_VEL
LIN {X 0,Y 192.705,Z 159.289,A -85,B 0,C 180,E1 -21936.348,E2 -21936.348} C_VEL
LIN {X 0,Y 192.731,Z 159.262,A -85,B 0,C 180,E1 -21941.457,E2 -21941.457} C_VEL
LIN {X 0,Y 192.772,Z 159.283,A -85,B 0,C 180,E1 -21945.214,E2 -21945.214} C_VEL
LIN {X 0,Y 192.98,Z 159.237,A -85,B 0,C 180,E1 -21949.508,E2 -21949.508} C_VEL
LIN {X 0,Y 193.061,Z 159.219,A -85,B 0,C 180,E1 -21951.627,E2 -21951.627} C_VEL
LIN {X 0,Y 193.264,Z 159.215,A -85,B 0,C 180,E1 -21957.916,E2 -21957.916} C_VEL
LIN {X 0,Y 193.443,Z 159.172,A -85,B 0,C 180,E1 -21960,E2 -21960} C_VEL
LIN {X 0,Y 192.978,Z 159.254,A -85,B 0,C 180,E1 -21964.177,E2 -21964.177} C_VEL
LIN {X 0,Y 193.068,Z 159.233,A -85,B 0,C 180,E1 -21968.372,E2 -21968.372} C_VEL
LIN {X 0,Y 192.852,Z 159.261,A -85,B 0,C 180,E1 -21972.63,E2 -21972.63} C_VEL
LIN {X 0,Y 192.757,Z 159.279,A -85,B 0,C 180,E1 -21976.959,E2 -21976.959} C_VEL
LIN {X 0,Y 192.635,Z 159.287,A -85,B 0,C 180,E1 -21981.397,E2 -21981.397} C_VEL
LIN {X 0,Y 192.663,Z 159.298,A -85,B 0,C 180,E1 -21984.225,E2 -21984.225} C_VEL
LIN {X 0,Y 192.649,Z 159.283,A -85,B 0,C 180,E1 -21988.892,E2 -21988.892} C_VEL
LIN {X 0,Y 192.597,Z 159.298,A -85,B 0,C 180,E1 -21993.186,E2 -21993.186} C_VEL
LIN {X 0,Y 192.55,Z 159.313,A -85,B 0,C 180,E1 -21998.352,E2 -21998.352} C_VEL
LIN {X 0,Y 192.486,Z 159.264,A -85,B 0,C 180,E1 -22003.095,E2 -22003.095} C_VEL
LIN {X 0,Y 192.488,Z 159.309,A -85,B 0,C 180,E1 -22006.905,E2 -22006.905} C_VEL
LIN {X 0,Y 192.558,Z 159.278,A -85,B 0,C 180,E1 -22011.651,E2 -22011.651} C_VEL
LIN {X 0,Y 192.62,Z 159.451,A -85,B 0,C 180,E1 -22012.856,E2 -22012.856} C_VEL
LIN {X 0,Y 193.72,Z 164.218,A -85,B 0,C 180,E1 -22015.917,E2 -22015.917} C_VEL
LIN {X 0,Y 195.41,Z 168.037,A -85,B 0,C 180,E1 -22016.543,E2 -22016.543} C_VEL
LIN {X 0,Y 201.875,Z 181.978,A -85,B 0,C 180,E1 -22018.314,E2 -22018.314} C_VEL
LIN {X 0,Y 205.553,Z 191.692,A -85,B 0,C 180,E1 -22019.329,E2 -22019.329} C_VEL
LIN {X 0,Y 208.289,Z 211.52,A -85,B 0,C 180,E1 -22020.544,E2 -22020.544} C_VEL
LIN {X 0,Y 207.287,Z 239.256,A -85,B 0,C 180,E1 -22021.496,E2 -22021.496} C_VEL
LIN {X 0,Y 206.42,Z 243.144,A -85,B 0,C 180,E1 -22021.567,E2 -22021.567} C_VEL
LIN {X 0,Y 203.331,Z 249.177,A -85,B 0,C 180,E1 -22021.548,E2 -22021.548} C_VEL
LIN {X 0,Y 200.088,Z 255.117,A -85,B 0,C 180,E1 -22021.593,E2 -22021.593} C_VEL
LIN {X 0,Y 199.046,Z 258.85,A -85,B 0,C 180,E1 -22021.876,E2 -22021.876} C_VEL
LIN {X 0,Y 197.62,Z 267.684,A -85,B 0,C 180,E1 -22022.882,E2 -22022.882} C_VEL
LIN {X 0,Y 195.81,Z 276.89,A -85,B 0,C 180,E1 -22024.255,E2 -22024.255} C_VEL
LIN {X 0,Y 193.203,Z 287.696,A -85,B 0,C 180,E1 -22026.414,E2 -22026.414} C_VEL
LIN {X 0,Y 191.116,Z 295.371,A -85,B 0,C 180,E1 -22028.425,E2 -22028.425} C_VEL
LIN {X 0,Y 189.251,Z 301.688,A -85,B 0,C 180,E1 -22030.475,E2 -22030.475} C_VEL
LIN {X 0,Y 187.6,Z 306.937,A -85,B 0,C 180,E1 -22032.561,E2 -22032.561} C_VEL
LIN {X 0,Y 186.315,Z 311.316,A -85,B 0,C 180,E1 -22034.69,E2 -22034.69} C_VEL
LIN {X 0,Y 184.763,Z 316.482,A -85,B 0,C 180,E1 -22037.925,E2 -22037.925} C_VEL
LIN {X 0,Y 183.737,Z 320.275,A -85,B 0,C 180,E1 -22041.2,E2 -22041.2} C_VEL
LIN {X 0,Y 183.312,Z 322.016,A -85,B 0,C 180,E1 -22043.396,E2 -22043.396} C_VEL
LIN {X 0,Y 183.026,Z 323.759,A -85,B 0,C 180,E1 -22046.726,E2 -22046.726} C_VEL
LIN {X 0,Y 183.072,Z 324.329,A -85,B 0,C 180,E1 -22050.001,E2 -22050.001} C_VEL
LIN {X 0,Y 183.031,Z 323.717,A -85,B 0,C 180,E1 -22053.301,E2 -22053.301} C_VEL
LIN {X 0,Y 183.314,Z 321.965,A -85,B 0,C 180,E1 -22056.605,E2 -22056.605} C_VEL
LIN {X 0,Y 183.984,Z 319.046,A -85,B 0,C 180,E1 -22059.899,E2 -22059.899} C_VEL
LIN {X 0,Y 184.723,Z 316.386,A -85,B 0,C 180,E1 -22062.079,E2 -22062.079} C_VEL
LIN {X 0,Y 186.313,Z 311.193,A -85,B 0,C 180,E1 -22065.311,E2 -22065.311} C_VEL
LIN {X 0,Y 188.368,Z 304.344,A -85,B 0,C 180,E1 -22068.49,E2 -22068.49} C_VEL
LIN {X 0,Y 190.608,Z 296.866,A -85,B 0,C 180,E1 -22071.07,E2 -22071.07} C_VEL
LIN {X 0,Y 192.668,Z 289.49,A -85,B 0,C 180,E1 -22073.088,E2 -22073.088} C_VEL
LIN {X 0,Y 194.62,Z 281.588,A -85,B 0,C 180,E1 -22074.822,E2 -22074.822} C_VEL
LIN {X 0,Y 196.586,Z 272.904,A -85,B 0,C 180,E1 -22076.321,E2 -22076.321} C_VEL
LIN {X 0,Y 198.505,Z 261.762,A -85,B 0,C 180,E1 -22077.79,E2 -22077.79} C_VEL
LIN {X 0,Y 199.977,Z 250.848,A -85,B 0,C 180,E1 -22078.753,E2 -22078.753} C_VEL
LIN {X 0,Y 200.833,Z 242.261,A -85,B 0,C 180,E1 -22079.264,E2 -22079.264} C_VEL
LIN {X 0,Y 201.978,Z 211.854,A -85,B 0,C 180,E1 -22080.382,E2 -22080.382} C_VEL
LIN {X 0,Y 199.258,Z 192.902,A -85,B 0,C 180,E1 -22081.62,E2 -22081.62} C_VEL
LIN {X 0,Y 193.931,Z 179.793,A -85,B 0,C 180,E1 -22083.154,E2 -22083.154} C_VEL
LIN {X 0,Y 187.853,Z 167.327,A -85,B 0,C 180,E1 -22084.933,E2 -22084.933} C_VEL
LIN {X 0,Y 186.476,Z 164.144,A -85,B 0,C 180,E1 -22085.498,E2 -22085.498} C_VEL
LIN {X 0,Y 185.542,Z 160.235,A -85,B 0,C 180,E1 -22088.161,E2 -22088.161} C_VEL
LIN {X 0,Y 185.459,Z 160.16,A -85,B 0,C 180,E1 -22093.945,E2 -22093.945} C_VEL
LIN {X 0,Y 185.471,Z 160.162,A -85,B 0,C 180,E1 -22099.276,E2 -22099.276} C_VEL
LIN {X 0,Y 185.508,Z 160.189,A -85,B 0,C 180,E1 -22102.712,E2 -22102.712} C_VEL
LIN {X 0,Y 185.548,Z 160.185,A -85,B 0,C 180,E1 -22107.976,E2 -22107.976} C_VEL
LIN {X 0,Y 185.584,Z 160.166,A -85,B 0,C 180,E1 -22110.576,E2 -22110.576} C_VEL
LIN {X 0,Y 185.59,Z 160.179,A -85,B 0,C 180,E1 -22115.383,E2 -22115.383} C_VEL
LIN {X 0,Y 185.677,Z 160.143,A -85,B 0,C 180,E1 -22121.133,E2 -22121.133} C_VEL
LIN {X 0,Y 185.722,Z 160.164,A -85,B 0,C 180,E1 -22124.64,E2 -22124.64} C_VEL
LIN {X 0,Y 185.891,Z 160.11,A -85,B 0,C 180,E1 -22129.418,E2 -22129.418} C_VEL
LIN {X 0,Y 185.954,Z 160.132,A -85,B 0,C 180,E1 -22133.49,E2 -22133.49} C_VEL
LIN {X 0,Y 186.209,Z 160.075,A -85,B 0,C 180,E1 -22137.837,E2 -22137.837} C_VEL
LIN {X 0,Y 186.407,Z 160.046,A -85,B 0,C 180,E1 -22140,E2 -22140} C_VEL
LIN {X 0,Y 185.928,Z 160.137,A -85,B 0,C 180,E1 -22144.336,E2 -22144.336} C_VEL
LIN {X 0,Y 186.012,Z 160.095,A -85,B 0,C 180,E1 -22148.693,E2 -22148.693} C_VEL
LIN {X 0,Y 185.767,Z 160.156,A -85,B 0,C 180,E1 -22153.12,E2 -22153.12} C_VEL
LIN {X 0,Y 185.693,Z 160.138,A -85,B 0,C 180,E1 -22157.625,E2 -22157.625} C_VEL
LIN {X 0,Y 185.599,Z 160.177,A -85,B 0,C 180,E1 -22162.251,E2 -22162.251} C_VEL
LIN {X 0,Y 185.565,Z 160.159,A -85,B 0,C 180,E1 -22167.032,E2 -22167.032} C_VEL
LIN {X 0,Y 185.581,Z 160.178,A -85,B 0,C 180,E1 -22169.493,E2 -22169.493} C_VEL
LIN {X 0,Y 185.502,Z 160.172,A -85,B 0,C 180,E1 -22174.632,E2 -22174.632} C_VEL
LIN {X 0,Y 185.508,Z 160.19,A -85,B 0,C 180,E1 -22177.313,E2 -22177.313} C_VEL
LIN {X 0,Y 185.473,Z 160.181,A -85,B 0,C 180,E1 -22180.725,E2 -22180.725} C_VEL
LIN {X 0,Y 185.481,Z 160.188,A -85,B 0,C 180,E1 -22183.951,E2 -22183.951} C_VEL
LIN {X 0,Y 185.486,Z 160.153,A -85,B 0,C 180,E1 -22189.271,E2 -22189.271} C_VEL
LIN {X 0,Y 185.592,Z 160.389,A -85,B 0,C 180,E1 -22194.224,E2 -22194.224} C_VEL
LIN {X 0,Y 185.85,Z 161.534,A -85,B 0,C 180,E1 -22194.646,E2 -22194.646} C_VEL
LIN {X 0,Y 187.529,Z 164.309,A -85,B 0,C 180,E1 -22195.16,E2 -22195.16} C_VEL
LIN {X 0,Y 193.086,Z 174.222,A -85,B 0,C 180,E1 -22196.74,E2 -22196.74} C_VEL
LIN {X 0,Y 199.251,Z 188.38,A -85,B 0,C 180,E1 -22198.491,E2 -22198.491} C_VEL
LIN {X 0,Y 202.308,Z 197.246,A -85,B 0,C 180,E1 -22199.383,E2 -22199.383} C_VEL
LIN {X 0,Y 202.581,Z 200.368,A -85,B 0,C 180,E1 -22199.555,E2 -22199.555} C_VEL
LIN {X 0,Y 201.018,Z 235.496,A -85,B 0,C 180,E1 -22200.788,E2 -22200.788} C_VEL
LIN {X 0,Y 200.081,Z 246.545,A -85,B 0,C 180,E1 -22201.485,E2 -22201.485} C_VEL
LIN {X 0,Y 198.616,Z 257.809,A -85,B 0,C 180,E1 -22202.612,E2 -22202.612} C_VEL
LIN {X 0,Y 197.054,Z 266.61,A -85,B 0,C 180,E1 -22203.809,E2 -22203.809} C_VEL
LIN {X 0,Y 195.323,Z 274.988,A -85,B 0,C 180,E1 -22205.273,E2 -22205.273} C_VEL
LIN {X 0,Y 193.34,Z 282.902,A -85,B 0,C 180,E1 -22206.997,E2 -22206.997} C_VEL
LIN {X 0,Y 191.318,Z 290.281,A -85,B 0,C 180,E1 -22209.012,E2 -22209.012} C_VEL
LIN {X 0,Y 189.157,Z 297.754,A -85,B 0,C 180,E1 -22211.59,E2 -22211.59} C_VEL
LIN {X 0,Y 186.937,Z 304.603,A -85,B 0,C 180,E1 -22214.741,E2 -22214.741} C_VEL
LIN {X 0,Y 185.317,Z 309.778,A -85,B 0,C 180,E1 -22217.96,E2 -22217.96} C_VEL
LIN {X 0,Y 184.49,Z 312.432,A -85,B 0,C 180,E1 -22220.129,E2 -22220.129} C_VEL
LIN {X 0,Y 183.687,Z 315.336,A -85,B 0,C 180,E1 -22223.408,E2 -22223.408} C_VEL
LIN {X 0,Y 183.337,Z 316.603,A -85,B 0,C 180,E1 -22225.602,E2 -22225.602} C_VEL
LIN {X 0,Y 183.131,Z 317.4,A -85,B 0,C 180,E1 -22227.8,E2 -22227.8} C_VEL
LIN {X 0,Y 183.114,Z 317.703,A -85,B 0,C 180,E1 -22229.999,E2 -22229.999} C_VEL
LIN {X 0,Y 183.13,Z 317.423,A -85,B 0,C 180,E1 -22232.199,E2 -22232.199} C_VEL
LIN {X 0,Y 183.396,Z 316.457,A -85,B 0,C 180,E1 -22234.89,E2 -22234.89} C_VEL
LIN {X 0,Y 184.133,Z 313.745,A -85,B 0,C 180,E1 -22238.781,E2 -22238.781} C_VEL
LIN {X 0,Y 185.29,Z 309.996,A -85,B 0,C 180,E1 -22242.041,E2 -22242.041} C_VEL
LIN {X 0,Y 186.904,Z 304.879,A -85,B 0,C 180,E1 -22245.26,E2 -22245.26} C_VEL
LIN {X 0,Y 188.683,Z 299.372,A -85,B 0,C 180,E1 -22247.896,E2 -22247.896} C_VEL
LIN {X 0,Y 190.786,Z 292.448,A -85,B 0,C 180,E1 -22250.484,E2 -22250.484} C_VEL
LIN {X 0,Y 193.019,Z 284.496,A -85,B 0,C 180,E1 -22252.759,E2 -22252.759} C_VEL
LIN {X 0,Y 194.968,Z 276.913,A -85,B 0,C 180,E1 -22254.49,E2 -22254.49} C_VEL
LIN {X 0,Y 196.718,Z 268.962,A -85,B 0,C 180,E1 -22255.953,E2 -22255.953} C_VEL
LIN {X 0,Y 198.255,Z 260.742,A -85,B 0,C 180,E1 -22257.155,E2 -22257.155} C_VEL
LIN {X 0,Y 199.522,Z 252.413,A -85,B 0,C 180,E1 -22258.105,E2 -22258.105} C_VEL
LIN {X 0,Y 200.587,Z 242.696,A -85,B 0,C 180,E1 -22258.929,E2 -22258.929} C_VEL
LIN {X 0,Y 201.295,Z 232.792,A -85,B 0,C 180,E1 -22259.48,E2 -22259.48} C_VEL
LIN {X 0,Y 202.627,Z 198.838,A -85,B 0,C 180,E1 -22260.662,E2 -22260.662} C_VEL
LIN {X 0,Y 201.673,Z 194.849,A -85,B 0,C 180,E1 -22260.986,E2 -22260.986} C_VEL
LIN {X 0,Y 196.629,Z 181.988,A -85,B 0,C 180,E1 -22262.42,E2 -22262.42} C_VEL
LIN {X 0,Y 191.459,Z 171.08,A -85,B 0,C 180,E1 -22263.894,E2 -22263.894} C_VEL
LIN {X 0,Y 187.136,Z 163.855,A -85,B 0,C 180,E1 -22265.124,E2 -22265.124} C_VEL
LIN {X 0,Y 185.728,Z 161.074,A -85,B 0,C 180,E1 -22265.626,E2 -22265.626} C_VEL
LIN {X 0,Y 185.559,Z 160.241,A -85,B 0,C 180,E1 -22266.144,E2 -22266.144} C_VEL
LIN {X 0,Y 185.483,Z 160.155,A -85,B 0,C 180,E1 -22270.729,E2 -22270.729} C_VEL
LIN {X 0,Y 185.478,Z 160.186,A -85,B 0,C 180,E1 -22276.048,E2 -22276.048} C_VEL
LIN {X 0,Y 185.467,Z 160.18,A -85,B 0,C 180,E1 -22279.895,E2 -22279.895} C_VEL
LIN {X 0,Y 185.506,Z 160.19,A -85,B 0,C 180,E1 -22282.711,E2 -22282.711} C_VEL
LIN {X 0,Y 185.546,Z 160.174,A -85,B 0,C 180,E1 -22287.975,E2 -22287.975} C_VEL
LIN {X 0,Y 185.581,Z 160.179,A -85,B 0,C 180,E1 -22290.575,E2 -22290.575} C_VEL
LIN {X 0,Y 185.587,Z 160.166,A -85,B 0,C 180,E1 -22295.382,E2 -22295.382} C_VEL
LIN {X 0,Y 185.606,Z 160.159,A -85,B 0,C 180,E1 -22300.075,E2 -22300.075} C_VEL
LIN {X 0,Y 185.724,Z 160.155,A -85,B 0,C 180,E1 -22304.639,E2 -22304.639} C_VEL
LIN {X 0,Y 185.923,Z 160.116,A -85,B 0,C 180,E1 -22309.359,E2 -22309.359} C_VEL
LIN {X 0,Y 185.961,Z 160.12,A -85,B 0,C 180,E1 -22313.49,E2 -22313.49} C_VEL
LIN {X 0,Y 186.208,Z 160.094,A -85,B 0,C 180,E1 -22317.837,E2 -22317.837} C_VEL
LIN {X 0,Y 186.406,Z 160.047,A -85,B 0,C 180,E1 -22320,E2 -22320} C_VEL
LIN {X 0,Y 185.926,Z 160.133,A -85,B 0,C 180,E1 -22324.335,E2 -22324.335} C_VEL
LIN {X 0,Y 186.013,Z 160.106,A -85,B 0,C 180,E1 -22328.692,E2 -22328.692} C_VEL
LIN {X 0,Y 185.764,Z 160.149,A -85,B 0,C 180,E1 -22333.12,E2 -22333.12} C_VEL
LIN {X 0,Y 185.689,Z 160.153,A -85,B 0,C 180,E1 -22337.625,E2 -22337.625} C_VEL
LIN {X 0,Y 185.596,Z 160.173,A -85,B 0,C 180,E1 -22342.251,E2 -22342.251} C_VEL
LIN {X 0,Y 185.561,Z 160.161,A -85,B 0,C 180,E1 -22347.032,E2 -22347.032} C_VEL
LIN {X 0,Y 185.578,Z 160.169,A -85,B 0,C 180,E1 -22349.493,E2 -22349.493} C_VEL
LIN {X 0,Y 185.498,Z 160.173,A -85,B 0,C 180,E1 -22354.632,E2 -22354.632} C_VEL
LIN {X 0,Y 185.505,Z 160.191,A -85,B 0,C 180,E1 -22357.313,E2 -22357.313} C_VEL
LIN {X 0,Y 185.469,Z 160.16,A -85,B 0,C 180,E1 -22360.725,E2 -22360.725} C_VEL
LIN {X 0,Y 185.456,Z 160.162,A -85,B 0,C 180,E1 -22366.056,E2 -22366.056} C_VEL
LIN {X 0,Y 185.52,Z 160.196,A -85,B 0,C 180,E1 -22371.662,E2 -22371.662} C_VEL
LIN {X 0,Y 186.381,Z 163.915,A -85,B 0,C 180,E1 -22374.317,E2 -22374.317} C_VEL
LIN {X 0,Y 187.239,Z 166.189,A -85,B 0,C 180,E1 -22374.796,E2 -22374.796} C_VEL
LIN {X 0,Y 191.595,Z 174.846,A -85,B 0,C 180,E1 -22376.09,E2 -22376.09} C_VEL
LIN {X 0,Y 196.857,Z 186.536,A -85,B 0,C 180,E1 -22377.605,E2 -22377.605} C_VEL
LIN {X 0,Y 199.729,Z 194.467,A -85,B 0,C 180,E1 -22378.452,E2 -22378.452} C_VEL
LIN {X 0,Y 202.127,Z 212.847,A -85,B 0,C 180,E1 -22379.61,E2 -22379.61} C_VEL
LIN {X 0,Y 200.888,Z 242.279,A -85,B 0,C 180,E1 -22380.674,E2 -22380.674} C_VEL
LIN {X 0,Y 199.806,Z 253.342,A -85,B 0,C 180,E1 -22381.365,E2 -22381.365} C_VEL
LIN {X 0,Y 199.046,Z 258.85,A -85,B 0,C 180,E1 -22381.876,E2 -22381.876} C_VEL
LIN {X 0,Y 197.682,Z 264.402,A -85,B 0,C 180,E1 -22382.379,E2 -22382.379} C_VEL
LIN {X 0,Y 193.565,Z 272.968,A -85,B 0,C 180,E1 -22383.158,E2 -22383.158} C_VEL
LIN {X 0,Y 189.103,Z 281.116,A -85,B 0,C 180,E1 -22384.206,E2 -22384.206} C_VEL
LIN {X 0,Y 187.232,Z 285.839,A -85,B 0,C 180,E1 -22385.127,E2 -22385.127} C_VEL
LIN {X 0,Y 185.069,Z 293.539,A -85,B 0,C 180,E1 -22387.093,E2 -22387.093} C_VEL
LIN {X 0,Y 183.034,Z 300.14,A -85,B 0,C 180,E1 -22389.196,E2 -22389.196} C_VEL
LIN {X 0,Y 181.276,Z 305.636,A -85,B 0,C 180,E1 -22391.347,E2 -22391.347} C_VEL
LIN {X 0,Y 179.451,Z 311.188,A -85,B 0,C 180,E1 -22394.089,E2 -22394.089} C_VEL
LIN {X 0,Y 177.798,Z 316.354,A -85,B 0,C 180,E1 -22397.444,E2 -22397.444} C_VEL
LIN {X 0,Y 176.717,Z 320.147,A -85,B 0,C 180,E1 -22400.847,E2 -22400.847} C_VEL
LIN {X 0,Y 176.252,Z 321.888,A -85,B 0,C 180,E1 -22403.13,E2 -22403.13} C_VEL
LIN {X 0,Y 175.946,Z 323.768,A -85,B 0,C 180,E1 -22406.964,E2 -22406.964} C_VEL
LIN {X 0,Y 175.984,Z 324.201,A -85,B 0,C 180,E1 -22410.001,E2 -22410.001} C_VEL
LIN {X 0,Y 175.928,Z 323.781,A -85,B 0,C 180,E1 -22412.919,E2 -22412.919} C_VEL
LIN {X 0,Y 176.252,Z 321.836,A -85,B 0,C 180,E1 -22416.871,E2 -22416.871} C_VEL
LIN {X 0,Y 176.994,Z 318.917,A -85,B 0,C 180,E1 -22420.294,E2 -22420.294} C_VEL
LIN {X 0,Y 177.763,Z 316.256,A -85,B 0,C 180,E1 -22422.56,E2 -22422.56} C_VEL
LIN {X 0,Y 179.447,Z 311.063,A -85,B 0,C 180,E1 -22425.912,E2 -22425.912} C_VEL
LIN {X 0,Y 181.634,Z 304.213,A -85,B 0,C 180,E1 -22429.202,E2 -22429.202} C_VEL
LIN {X 0,Y 184.006,Z 296.735,A -85,B 0,C 180,E1 -22431.864,E2 -22431.864} C_VEL
LIN {X 0,Y 186.149,Z 289.358,A -85,B 0,C 180,E1 -22433.946,E2 -22433.946} C_VEL
LIN {X 0,Y 188.215,Z 281.456,A -85,B 0,C 180,E1 -22435.727,E2 -22435.727} C_VEL
LIN {X 0,Y 190.438,Z 271.876,A -85,B 0,C 180,E1 -22437.417,E2 -22437.417} C_VEL
LIN {X 0,Y 192.494,Z 260.053,A -85,B 0,C 180,E1 -22438.932,E2 -22438.932} C_VEL
LIN {X 0,Y 193.796,Z 250.701,A -85,B 0,C 180,E1 -22439.761,E2 -22439.761} C_VEL
LIN {X 0,Y 194.736,Z 240.817,A -85,B 0,C 180,E1 -22440.349,E2 -22440.349} C_VEL
LIN {X 0,Y 195.874,Z 212.707,A -85,B 0,C 180,E1 -22441.392,E2 -22441.392} C_VEL
LIN {X 0,Y 193.493,Z 195.549,A -85,B 0,C 180,E1 -22442.557,E2 -22442.557} C_VEL
LIN {X 0,Y 188.323,Z 182.863,A -85,B 0,C 180,E1 -22444.131,E2 -22444.131} C_VEL
LIN {X 0,Y 182.767,Z 171.269,A -85,B 0,C 180,E1 -22445.86,E2 -22445.86} C_VEL
LIN {X 0,Y 179.276,Z 164.222,A -85,B 0,C 180,E1 -22447.094,E2 -22447.094} C_VEL
LIN {X 0,Y 178.795,Z 162.402,A -85,B 0,C 180,E1 -22448.173,E2 -22448.173} C_VEL
LIN {X 0,Y 178.448,Z 161.071,A -85,B 0,C 180,E1 -22449.426,E2 -22449.426} C_VEL
LIN {X 0,Y 178.393,Z 161.021,A -85,B 0,C 180,E1 -22455.165,E2 -22455.165} C_VEL
LIN {X 0,Y 178.403,Z 161.026,A -85,B 0,C 180,E1 -22458.46,E2 -22458.46} C_VEL
LIN {X 0,Y 178.424,Z 161.06,A -85,B 0,C 180,E1 -22463.784,E2 -22463.784} C_VEL
LIN {X 0,Y 178.488,Z 161.052,A -85,B 0,C 180,E1 -22466.547,E2 -22466.547} C_VEL
LIN {X 0,Y 178.525,Z 161.051,A -85,B 0,C 180,E1 -22470.007,E2 -22470.007} C_VEL
LIN {X 0,Y 178.536,Z 161.053,A -85,B 0,C 180,E1 -22474.876,E2 -22474.876} C_VEL
LIN {X 0,Y 178.625,Z 161.019,A -85,B 0,C 180,E1 -22480.784,E2 -22480.784} C_VEL
LIN {X 0,Y 178.664,Z 161.04,A -85,B 0,C 180,E1 -22484.017,E2 -22484.017} C_VEL
LIN {X 0,Y 178.836,Z 160.987,A -85,B 0,C 180,E1 -22489.256,E2 -22489.256} C_VEL
LIN {X 0,Y 178.917,Z 161.009,A -85,B 0,C 180,E1 -22493.233,E2 -22493.233} C_VEL
LIN {X 0,Y 179.155,Z 160.953,A -85,B 0,C 180,E1 -22497.752,E2 -22497.752} C_VEL
LIN {X 0,Y 179.37,Z 160.921,A -85,B 0,C 180,E1 -22500,E2 -22500} C_VEL
LIN {X 0,Y 178.876,Z 161.015,A -85,B 0,C 180,E1 -22504.507,E2 -22504.507} C_VEL
LIN {X 0,Y 178.941,Z 160.974,A -85,B 0,C 180,E1 -22509.039,E2 -22509.039} C_VEL
LIN {X 0,Y 178.69,Z 161.04,A -85,B 0,C 180,E1 -22513.65,E2 -22513.65} C_VEL
LIN {X 0,Y 178.652,Z 161.013,A -85,B 0,C 180,E1 -22518.344,E2 -22518.344} C_VEL
LIN {X 0,Y 178.514,Z 161.059,A -85,B 0,C 180,E1 -22523.185,E2 -22523.185} C_VEL
LIN {X 0,Y 178.489,Z 161.047,A -85,B 0,C 180,E1 -22528.197,E2 -22528.197} C_VEL
LIN {X 0,Y 178.503,Z 161.062,A -85,B 0,C 180,E1 -22530.786,E2 -22530.786} C_VEL
LIN {X 0,Y 178.487,Z 161.044,A -85,B 0,C 180,E1 -22534.219,E2 -22534.219} C_VEL
LIN {X 0,Y 178.397,Z 161.063,A -85,B 0,C 180,E1 -22539.074,E2 -22539.074} C_VEL
LIN {X 0,Y 178.408,Z 161.072,A -85,B 0,C 180,E1 -22542.043,E2 -22542.043} C_VEL
LIN {X 0,Y 178.4,Z 161.045,A -85,B 0,C 180,E1 -22545.162,E2 -22545.162} C_VEL
LIN {X 0,Y 178.411,Z 161.025,A -85,B 0,C 180,E1 -22548.457,E2 -22548.457} C_VEL
LIN {X 0,Y 178.511,Z 161.251,A -85,B 0,C 180,E1 -22552.601,E2 -22552.601} C_VEL
LIN {X 0,Y 178.803,Z 162.415,A -85,B 0,C 180,E1 -22553.063,E2 -22553.063} C_VEL
LIN {X 0,Y 180.371,Z 165.06,A -85,B 0,C 180,E1 -22553.589,E2 -22553.589} C_VEL
LIN {X 0,Y 187.235,Z 176.803,A -85,B 0,C 180,E1 -22555.669,E2 -22555.669} C_VEL
LIN {X 0,Y 192.815,Z 189.411,A -85,B 0,C 180,E1 -22557.349,E2 -22557.349} C_VEL
LIN {X 0,Y 196.399,Z 199.468,A -85,B 0,C 180,E1 -22558.445,E2 -22558.445} C_VEL
LIN {X 0,Y 195.74,Z 217.971,A -85,B 0,C 180,E1 -22559.105,E2 -22559.105} C_VEL
LIN {X 0,Y 194.744,Z 237.696,A -85,B 0,C 180,E1 -22559.869,E2 -22559.869} C_VEL
LIN {X 0,Y 193.509,Z 249.549,A -85,B 0,C 180,E1 -22560.738,E2 -22560.738} C_VEL
LIN {X 0,Y 192.035,Z 259.813,A -85,B 0,C 180,E1 -22561.888,E2 -22561.888} C_VEL
LIN {X 0,Y 190.403,Z 268.242,A -85,B 0,C 180,E1 -22563.117,E2 -22563.117} C_VEL
LIN {X 0,Y 188.599,Z 276.349,A -85,B 0,C 180,E1 -22564.625,E2 -22564.625} C_VEL
LIN {X 0,Y 186.56,Z 284.053,A -85,B 0,C 180,E1 -22566.405,E2 -22566.405} C_VEL
LIN {X 0,Y 184.247,Z 292.109,A -85,B 0,C 180,E1 -22568.753,E2 -22568.753} C_VEL
LIN {X 0,Y 182.008,Z 299.161,A -85,B 0,C 180,E1 -22571.423,E2 -22571.423} C_VEL
LIN {X 0,Y 180.103,Z 304.732,A -85,B 0,C 180,E1 -22574.147,E2 -22574.147} C_VEL
LIN {X 0,Y 178.382,Z 309.908,A -85,B 0,C 180,E1 -22577.485,E2 -22577.485} C_VEL
LIN {X 0,Y 177.497,Z 312.561,A -85,B 0,C 180,E1 -22579.736,E2 -22579.736} C_VEL
LIN {X 0,Y 176.64,Z 315.465,A -85,B 0,C 180,E1 -22583.144,E2 -22583.144} C_VEL
LIN {X 0,Y 176.262,Z 316.731,A -85,B 0,C 180,E1 -22585.426,E2 -22585.426} C_VEL
LIN {X 0,Y 176.036,Z 317.529,A -85,B 0,C 180,E1 -22587.711,E2 -22587.711} C_VEL
LIN {X 0,Y 176.026,Z 317.831,A -85,B 0,C 180,E1 -22589.999,E2 -22589.999} C_VEL
LIN {X 0,Y 176.035,Z 317.552,A -85,B 0,C 180,E1 -22592.288,E2 -22592.288} C_VEL
LIN {X 0,Y 176.262,Z 316.8,A -85,B 0,C 180,E1 -22594.573,E2 -22594.573} C_VEL
LIN {X 0,Y 176.575,Z 315.582,A -85,B 0,C 180,E1 -22596.857,E2 -22596.857} C_VEL
LIN {X 0,Y 177.49,Z 312.725,A -85,B 0,C 180,E1 -22600.263,E2 -22600.263} C_VEL
LIN {X 0,Y 178.356,Z 310.123,A -85,B 0,C 180,E1 -22602.516,E2 -22602.516} C_VEL
LIN {X 0,Y 180.074,Z 305.006,A -85,B 0,C 180,E1 -22605.854,E2 -22605.854} C_VEL
LIN {X 0,Y 181.959,Z 299.498,A -85,B 0,C 180,E1 -22608.581,E2 -22608.581} C_VEL
LIN {X 0,Y 184.154,Z 292.574,A -85,B 0,C 180,E1 -22611.257,E2 -22611.257} C_VEL
LIN {X 0,Y 186.513,Z 284.621,A -85,B 0,C 180,E1 -22613.6,E2 -22613.6} C_VEL
LIN {X 0,Y 188.546,Z 277.037,A -85,B 0,C 180,E1 -22615.382,E2 -22615.382} C_VEL
LIN {X 0,Y 190.379,Z 269.085,A -85,B 0,C 180,E1 -22616.885,E2 -22616.885} C_VEL
LIN {X 0,Y 191.981,Z 260.864,A -85,B 0,C 180,E1 -22618.12,E2 -22618.12} C_VEL
LIN {X 0,Y 193.284,Z 252.534,A -85,B 0,C 180,E1 -22619.097,E2 -22619.097} C_VEL
LIN {X 0,Y 194.402,Z 243.01,A -85,B 0,C 180,E1 -22619.924,E2 -22619.924} C_VEL
LIN {X 0,Y 195.059,Z 234.268,A -85,B 0,C 180,E1 -22620.442,E2 -22620.442} C_VEL
LIN {X 0,Y 196.516,Z 199.645,A -85,B 0,C 180,E1 -22621.694,E2 -22621.694} C_VEL
LIN {X 0,Y 192.369,Z 188.195,A -85,B 0,C 180,E1 -22622.962,E2 -22622.962} C_VEL
LIN {X 0,Y 187.064,Z 176.454,A -85,B 0,C 180,E1 -22624.561,E2 -22624.561} C_VEL
LIN {X 0,Y 180.282,Z 164.909,A -85,B 0,C 180,E1 -22626.626,E2 -22626.626} C_VEL
LIN {X 0,Y 178.688,Z 162.058,A -85,B 0,C 180,E1 -22627.197,E2 -22627.197} C_VEL
LIN {X 0,Y 178.46,Z 161.125,A -85,B 0,C 180,E1 -22627.724,E2 -22627.724} C_VEL
LIN {X 0,Y 178.401,Z 161.024,A -85,B 0,C 180,E1 -22632.043,E2 -22632.043} C_VEL
LIN {X 0,Y 178.4,Z 161.046,A -85,B 0,C 180,E1 -22635.161,E2 -22635.161} C_VEL
LIN {X 0,Y 178.407,Z 161.068,A -85,B 0,C 180,E1 -22638.457,E2 -22638.457} C_VEL
LIN {X 0,Y 178.422,Z 161.071,A -85,B 0,C 180,E1 -22643.783,E2 -22643.783} C_VEL
LIN {X 0,Y 178.486,Z 161.044,A -85,B 0,C 180,E1 -22646.546,E2 -22646.546} C_VEL
LIN {X 0,Y 178.522,Z 161.06,A -85,B 0,C 180,E1 -22650.006,E2 -22650.006} C_VEL
LIN {X 0,Y 178.534,Z 161.038,A -85,B 0,C 180,E1 -22654.875,E2 -22654.875} C_VEL
LIN {X 0,Y 178.622,Z 161.021,A -85,B 0,C 180,E1 -22660.783,E2 -22660.783} C_VEL
LIN {X 0,Y 178.665,Z 161.027,A -85,B 0,C 180,E1 -22664.017,E2 -22664.017} C_VEL
LIN {X 0,Y 178.86,Z 160.996,A -85,B 0,C 180,E1 -22669.21,E2 -22669.21} C_VEL
LIN {X 0,Y 178.925,Z 160.991,A -85,B 0,C 180,E1 -22673.232,E2 -22673.232} C_VEL
LIN {X 0,Y 179.154,Z 160.972,A -85,B 0,C 180,E1 -22677.752,E2 -22677.752} C_VEL
LIN {X 0,Y 179.369,Z 160.922,A -85,B 0,C 180,E1 -22680,E2 -22680} C_VEL
LIN {X 0,Y 178.875,Z 161.013,A -85,B 0,C 180,E1 -22684.507,E2 -22684.507} C_VEL
LIN {X 0,Y 178.963,Z 160.979,A -85,B 0,C 180,E1 -22689.037,E2 -22689.037} C_VEL
LIN {X 0,Y 178.686,Z 161.033,A -85,B 0,C 180,E1 -22693.65,E2 -22693.65} C_VEL
LIN {X 0,Y 178.649,Z 161.021,A -85,B 0,C 180,E1 -22698.344,E2 -22698.344} C_VEL
LIN {X 0,Y 178.51,Z 161.061,A -85,B 0,C 180,E1 -22703.185,E2 -22703.185} C_VEL
LIN {X 0,Y 178.485,Z 161.041,A -85,B 0,C 180,E1 -22708.197,E2 -22708.197} C_VEL
LIN {X 0,Y 178.5,Z 161.062,A -85,B 0,C 180,E1 -22710.786,E2 -22710.786} C_VEL
LIN {X 0,Y 178.484,Z 161.047,A -85,B 0,C 180,E1 -22714.22,E2 -22714.22} C_VEL
LIN {X 0,Y 178.394,Z 161.07,A -85,B 0,C 180,E1 -22719.075,E2 -22719.075} C_VEL
LIN {X 0,Y 178.395,Z 161.02,A -85,B 0,C 180,E1 -22722.046,E2 -22722.046} C_VEL
LIN {X 0,Y 178.391,Z 161.026,A -85,B 0,C 180,E1 -22725.165,E2 -22725.165} C_VEL
LIN {X 0,Y 178.477,Z 161.183,A -85,B 0,C 180,E1 -22730.766,E2 -22730.766} C_VEL
LIN {X 0,Y 179.149,Z 163.952,A -85,B 0,C 180,E1 -22732.707,E2 -22732.707} C_VEL
LIN {X 0,Y 181.003,Z 167.805,A -85,B 0,C 180,E1 -22733.475,E2 -22733.475} C_VEL
LIN {X 0,Y 187.422,Z 180.829,A -85,B 0,C 180,E1 -22735.504,E2 -22735.504} C_VEL
LIN {X 0,Y 192.142,Z 191.884,A -85,B 0,C 180,E1 -22736.946,E2 -22736.946} C_VEL
LIN {X 0,Y 193.882,Z 196.822,A -85,B 0,C 180,E1 -22737.491,E2 -22737.491} C_VEL
LIN {X 0,Y 196.003,Z 213.532,A -85,B 0,C 180,E1 -22738.588,E2 -22738.588} C_VEL
LIN {X 0,Y 194.738,Z 242.166,A -85,B 0,C 180,E1 -22739.653,E2 -22739.653} C_VEL
LIN {X 0,Y 193.605,Z 253.214,A -85,B 0,C 180,E1 -22740.357,E2 -22740.357} C_VEL
LIN {X 0,Y 191.825,Z 264.823,A -85,B 0,C 180,E1 -22741.557,E2 -22741.557} C_VEL
LIN {X 0,Y 190.102,Z 273.605,A -85,B 0,C 180,E1 -22742.798,E2 -22742.798} C_VEL
LIN {X 0,Y 188.23,Z 281.771,A -85,B 0,C 180,E1 -22744.276,E2 -22744.276} C_VEL
LIN {X 0,Y 187.232,Z 285.839,A -85,B 0,C 180,E1 -22745.127,E2 -22745.127} C_VEL
LIN {X 0,Y 185.324,Z 290.39,A -85,B 0,C 180,E1 -22746.15,E2 -22746.15} C_VEL
LIN {X 0,Y 180.553,Z 297.244,A -85,B 0,C 180,E1 -22747.822,E2 -22747.822} C_VEL
LIN {X 0,Y 175.823,Z 303.483,A -85,B 0,C 180,E1 -22749.787,E2 -22749.787} C_VEL
LIN {X 0,Y 174.023,Z 306.867,A -85,B 0,C 180,E1 -22751.247,E2 -22751.247} C_VEL
LIN {X 0,Y 172.61,Z 311.061,A -85,B 0,C 180,E1 -22753.441,E2 -22753.441} C_VEL
LIN {X 0,Y 170.848,Z 316.226,A -85,B 0,C 180,E1 -22756.924,E2 -22756.924} C_VEL
LIN {X 0,Y 169.699,Z 320.02,A -85,B 0,C 180,E1 -22760.465,E2 -22760.465} C_VEL
LIN {X 0,Y 169.188,Z 321.76,A -85,B 0,C 180,E1 -22762.842,E2 -22762.842} C_VEL
LIN {X 0,Y 168.937,Z 323.006,A -85,B 0,C 180,E1 -22765.228,E2 -22765.228} C_VEL
LIN {X 0,Y 168.857,Z 323.78,A -85,B 0,C 180,E1 -22767.615,E2 -22767.615} C_VEL
LIN {X 0,Y 168.884,Z 324.072,A -85,B 0,C 180,E1 -22770.001,E2 -22770.001} C_VEL
LIN {X 0,Y 168.852,Z 323.733,A -85,B 0,C 180,E1 -22772.654,E2 -22772.654} C_VEL
LIN {X 0,Y 168.937,Z 322.974,A -85,B 0,C 180,E1 -22774.773,E2 -22774.773} C_VEL
LIN {X 0,Y 169.186,Z 321.706,A -85,B 0,C 180,E1 -22777.159,E2 -22777.159} C_VEL
LIN {X 0,Y 169.992,Z 318.787,A -85,B 0,C 180,E1 -22780.723,E2 -22780.723} C_VEL
LIN {X 0,Y 170.816,Z 316.126,A -85,B 0,C 180,E1 -22783.079,E2 -22783.079} C_VEL
LIN {X 0,Y 172.606,Z 310.933,A -85,B 0,C 180,E1 -22786.561,E2 -22786.561} C_VEL
LIN {X 0,Y 174.941,Z 304.083,A -85,B 0,C 180,E1 -22789.967,E2 -22789.967} C_VEL
LIN {X 0,Y 177.441,Z 296.604,A -85,B 0,C 180,E1 -22792.717,E2 -22792.717} C_VEL
LIN {X 0,Y 179.666,Z 289.226,A -85,B 0,C 180,E1 -22794.867,E2 -22794.867} C_VEL
LIN {X 0,Y 181.853,Z 281.324,A -85,B 0,C 180,E1 -22796.697,E2 -22796.697} C_VEL
LIN {X 0,Y 184.229,Z 271.448,A -85,B 0,C 180,E1 -22798.484,E2 -22798.484} C_VEL
LIN {X 0,Y 186.317,Z 259.917,A -85,B 0,C 180,E1 -22799.987,E2 -22799.987} C_VEL
LIN {X 0,Y 187.67,Z 250.562,A -85,B 0,C 180,E1 -22800.836,E2 -22800.836} C_VEL
LIN {X 0,Y 188.645,Z 240.673,A -85,B 0,C 180,E1 -22801.438,E2 -22801.438} C_VEL
LIN {X 0,Y 189.786,Z 213.521,A -85,B 0,C 180,E1 -22802.478,E2 -22802.478} C_VEL
LIN {X 0,Y 187.685,Z 197.987,A -85,B 0,C 180,E1 -22803.58,E2 -22803.58} C_VEL
LIN {X 0,Y 182.99,Z 186.344,A -85,B 0,C 180,E1 -22805.1,E2 -22805.1} C_VEL
LIN {X 0,Y 177.07,Z 173.901,A -85,B 0,C 180,E1 -22807.066,E2 -22807.066} C_VEL
LIN {X 0,Y 173.38,Z 167.075,A -85,B 0,C 180,E1 -22808.339,E2 -22808.339} C_VEL
LIN {X 0,Y 171.893,Z 163.877,A -85,B 0,C 180,E1 -22809.029,E2 -22809.029} C_VEL
LIN {X 0,Y 171.388,Z 162.025,A -85,B 0,C 180,E1 -22810.416,E2 -22810.416} C_VEL
LIN {X 0,Y 171.32,Z 161.895,A -85,B 0,C 180,E1 -22815.783,E2 -22815.783} C_VEL
LIN {X 0,Y 171.359,Z 161.951,A -85,B 0,C 180,E1 -22821.193,E2 -22821.193} C_VEL
LIN {X 0,Y 171.4,Z 161.928,A -85,B 0,C 180,E1 -22825.093,E2 -22825.093} C_VEL
LIN {X 0,Y 171.45,Z 161.925,A -85,B 0,C 180,E1 -22830.535,E2 -22830.535} C_VEL
LIN {X 0,Y 171.46,Z 161.94,A -85,B 0,C 180,E1 -22835.802,E2 -22835.802} C_VEL
LIN {X 0,Y 171.581,Z 161.896,A -85,B 0,C 180,E1 -22840.872,E2 -22840.872} C_VEL
LIN {X 0,Y 171.593,Z 161.921,A -85,B 0,C 180,E1 -22845.774,E2 -22845.774} C_VEL
LIN {X 0,Y 171.852,Z 161.86,A -85,B 0,C 180,E1 -22850.585,E2 -22850.585} C_VEL
LIN {X 0,Y 171.82,Z 161.893,A -85,B 0,C 180,E1 -22855.308,E2 -22855.308} C_VEL
LIN {X 0,Y 172.333,Z 161.797,A -85,B 0,C 180,E1 -22860,E2 -22860} C_VEL
LIN {X 0,Y 171.825,Z 161.893,A -85,B 0,C 180,E1 -22864.693,E2 -22864.693} C_VEL
LIN {X 0,Y 171.876,Z 161.854,A -85,B 0,C 180,E1 -22869.414,E2 -22869.414} C_VEL
LIN {X 0,Y 171.612,Z 161.919,A -85,B 0,C 180,E1 -22874.224,E2 -22874.224} C_VEL
LIN {X 0,Y 171.547,Z 161.902,A -85,B 0,C 180,E1 -22879.562,E2 -22879.562} C_VEL
LIN {X 0,Y 171.471,Z 161.914,A -85,B 0,C 180,E1 -22885.616,E2 -22885.616} C_VEL
LIN {X 0,Y 171.461,Z 161.941,A -85,B 0,C 180,E1 -22890.596,E2 -22890.596} C_VEL
LIN {X 0,Y 171.395,Z 161.93,A -85,B 0,C 180,E1 -22895.035,E2 -22895.035} C_VEL
LIN {X 0,Y 171.359,Z 161.941,A -85,B 0,C 180,E1 -22898.807,E2 -22898.807} C_VEL
LIN {X 0,Y 171.329,Z 161.941,A -85,B 0,C 180,E1 -22904.215,E2 -22904.215} C_VEL
LIN {X 0,Y 171.345,Z 161.907,A -85,B 0,C 180,E1 -22908.984,E2 -22908.984} C_VEL
LIN {X 0,Y 171.427,Z 162.282,A -85,B 0,C 180,E1 -22910.927,E2 -22910.927} C_VEL
LIN {X 0,Y 171.804,Z 163.575,A -85,B 0,C 180,E1 -22911.346,E2 -22911.346} C_VEL
LIN {X 0,Y 173.49,Z 166.142,A -85,B 0,C 180,E1 -22911.941,E2 -22911.941} C_VEL
LIN {X 0,Y 180.52,Z 177.775,A -85,B 0,C 180,E1 -22914.238,E2 -22914.238} C_VEL
LIN {X 0,Y 184.513,Z 185.896,A -85,B 0,C 180,E1 -22915.509,E2 -22915.509} C_VEL
LIN {X 0,Y 189.474,Z 198.398,A -85,B 0,C 180,E1 -22917.094,E2 -22917.094} C_VEL
LIN {X 0,Y 190.45,Z 201.199,A -85,B 0,C 180,E1 -22917.408,E2 -22917.408} C_VEL
LIN {X 0,Y 188.791,Z 235.109,A -85,B 0,C 180,E1 -22918.65,E2 -22918.65} C_VEL
LIN {X 0,Y 187.918,Z 245.31,A -85,B 0,C 180,E1 -22919.309,E2 -22919.309} C_VEL
LIN {X 0,Y 186.534,Z 255.847,A -85,B 0,C 180,E1 -22920.327,E2 -22920.327} C_VEL
LIN {X 0,Y 184.457,Z 266.876,A -85,B 0,C 180,E1 -22921.868,E2 -22921.868} C_VEL
LIN {X 0,Y 182.55,Z 275.252,A -85,B 0,C 180,E1 -22923.413,E2 -22923.413} C_VEL
LIN {X 0,Y 180.356,Z 283.165,A -85,B 0,C 180,E1 -22925.234,E2 -22925.234} C_VEL
LIN {X 0,Y 178.14,Z 290.543,A -85,B 0,C 180,E1 -22927.377,E2 -22927.377} C_VEL
LIN {X 0,Y 175.725,Z 298.016,A -85,B 0,C 180,E1 -22930.126,E2 -22930.126} C_VEL
LIN {X 0,Y 173.282,Z 304.863,A -85,B 0,C 180,E1 -22933.506,E2 -22933.506} C_VEL
LIN {X 0,Y 171.445,Z 310.038,A -85,B 0,C 180,E1 -22936.97,E2 -22936.97} C_VEL
LIN {X 0,Y 170.525,Z 312.691,A -85,B 0,C 180,E1 -22939.311,E2 -22939.311} C_VEL
LIN {X 0,Y 169.591,Z 315.594,A -85,B 0,C 180,E1 -22942.858,E2 -22942.858} C_VEL
LIN {X 0,Y 169.108,Z 317.123,A -85,B 0,C 180,E1 -22945.888,E2 -22945.888} C_VEL
LIN {X 0,Y 168.941,Z 317.959,A -85,B 0,C 180,E1 -22949.999,E2 -22949.999} C_VEL
LIN {X 0,Y 169.108,Z 317.191,A -85,B 0,C 180,E1 -22954.111,E2 -22954.111} C_VEL
LIN {X 0,Y 169.531,Z 315.71,A -85,B 0,C 180,E1 -22957.144,E2 -22957.144} C_VEL
LIN {X 0,Y 170.519,Z 312.852,A -85,B 0,C 180,E1 -22960.688,E2 -22960.688} C_VEL
LIN {X 0,Y 171.415,Z 310.251,A -85,B 0,C 180,E1 -22963.032,E2 -22963.032} C_VEL
LIN {X 0,Y 173.256,Z 305.133,A -85,B 0,C 180,E1 -22966.495,E2 -22966.495} C_VEL
LIN {X 0,Y 175.236,Z 299.625,A -85,B 0,C 180,E1 -22969.321,E2 -22969.321} C_VEL
LIN {X 0,Y 177.567,Z 292.699,A -85,B 0,C 180,E1 -22972.086,E2 -22972.086} C_VEL
LIN {X 0,Y 180.037,Z 284.746,A -85,B 0,C 180,E1 -22974.504,E2 -22974.504} C_VEL
LIN {X 0,Y 182.176,Z 277.161,A -85,B 0,C 180,E1 -22976.336,E2 -22976.336} C_VEL
LIN {X 0,Y 184.08,Z 269.209,A -85,B 0,C 180,E1 -22977.884,E2 -22977.884} C_VEL
LIN {X 0,Y 185.764,Z 260.986,A -85,B 0,C 180,E1 -22979.149,E2 -22979.149} C_VEL
LIN {X 0,Y 187.189,Z 252.217,A -85,B 0,C 180,E1 -22980.197,E2 -22980.197} C_VEL
LIN {X 0,Y 188.251,Z 243.469,A -85,B 0,C 180,E1 -22980.975,E2 -22980.975} C_VEL
LIN {X 0,Y 188.979,Z 234.399,A -85,B 0,C 180,E1 -22981.53,E2 -22981.53} C_VEL
LIN {X 0,Y 190.52,Z 201.19,A -85,B 0,C 180,E1 -22982.751,E2 -22982.751} C_VEL
LIN {X 0,Y 185.753,Z 188.671,A -85,B 0,C 180,E1 -22984.279,E2 -22984.279} C_VEL
LIN {X 0,Y 181.235,Z 179.014,A -85,B 0,C 180,E1 -22985.723,E2 -22985.723} C_VEL
LIN {X 0,Y 175.269,Z 169.029,A -85,B 0,C 180,E1 -22987.649,E2 -22987.649} C_VEL
LIN {X 0,Y 173.493,Z 166.158,A -85,B 0,C 180,E1 -22988.253,E2 -22988.253} C_VEL
LIN {X 0,Y 171.835,Z 163.662,A -85,B 0,C 180,E1 -22988.836,E2 -22988.836} C_VEL
LIN {X 0,Y 171.456,Z 162.454,A -85,B 0,C 180,E1 -22989.154,E2 -22989.154} C_VEL
LIN {X 0,Y 171.355,Z 161.962,A -85,B 0,C 180,E1 -22989.811,E2 -22989.811} C_VEL
LIN {X 0,Y 171.324,Z 161.912,A -85,B 0,C 180,E1 -22994.215,E2 -22994.215} C_VEL
LIN {X 0,Y 171.338,Z 161.943,A -85,B 0,C 180,E1 -22998.982,E2 -22998.982} C_VEL
LIN {X 0,Y 171.386,Z 161.944,A -85,B 0,C 180,E1 -23002.04,E2 -23002.04} C_VEL
LIN {X 0,Y 171.398,Z 161.931,A -85,B 0,C 180,E1 -23005.092,E2 -23005.092} C_VEL
LIN {X 0,Y 171.449,Z 161.939,A -85,B 0,C 180,E1 -23010.534,E2 -23010.534} C_VEL
LIN {X 0,Y 171.457,Z 161.928,A -85,B 0,C 180,E1 -23015.801,E2 -23015.801} C_VEL
LIN {X 0,Y 171.578,Z 161.896,A -85,B 0,C 180,E1 -23020.871,E2 -23020.871} C_VEL
LIN {X 0,Y 171.609,Z 161.92,A -85,B 0,C 180,E1 -23025.775,E2 -23025.775} C_VEL
LIN {X 0,Y 171.873,Z 161.854,A -85,B 0,C 180,E1 -23030.586,E2 -23030.586} C_VEL
LIN {X 0,Y 171.823,Z 161.893,A -85,B 0,C 180,E1 -23035.307,E2 -23035.307} C_VEL
LIN {X 0,Y 172.332,Z 161.797,A -85,B 0,C 180,E1 -23040,E2 -23040} C_VEL
LIN {X 0,Y 171.824,Z 161.892,A -85,B 0,C 180,E1 -23044.692,E2 -23044.692} C_VEL
LIN {X 0,Y 171.891,Z 161.855,A -85,B 0,C 180,E1 -23049.413,E2 -23049.413} C_VEL
LIN {X 0,Y 171.609,Z 161.92,A -85,B 0,C 180,E1 -23054.224,E2 -23054.224} C_VEL
LIN {X 0,Y 171.543,Z 161.9,A -85,B 0,C 180,E1 -23059.562,E2 -23059.562} C_VEL
LIN {X 0,Y 171.468,Z 161.927,A -85,B 0,C 180,E1 -23065.616,E2 -23065.616} C_VEL
LIN {X 0,Y 171.457,Z 161.938,A -85,B 0,C 180,E1 -23070.596,E2 -23070.596} C_VEL
LIN {X 0,Y 171.391,Z 161.929,A -85,B 0,C 180,E1 -23075.035,E2 -23075.035} C_VEL
LIN {X 0,Y 171.356,Z 161.949,A -85,B 0,C 180,E1 -23078.808,E2 -23078.808} C_VEL
LIN {X 0,Y 171.318,Z 161.896,A -85,B 0,C 180,E1 -23084.218,E2 -23084.218} C_VEL
LIN {X 0,Y 171.415,Z 162.094,A -85,B 0,C 180,E1 -23089.593,E2 -23089.593} C_VEL
LIN {X 0,Y 171.866,Z 163.791,A -85,B 0,C 180,E1 -23090.83,E2 -23090.83} C_VEL
LIN {X 0,Y 173.703,Z 167.547,A -85,B 0,C 180,E1 -23091.664,E2 -23091.664} C_VEL
LIN {X 0,Y 179.57,Z 178.896,A -85,B 0,C 180,E1 -23093.677,E2 -23093.677} C_VEL
LIN {X 0,Y 185.453,Z 191.991,A -85,B 0,C 180,E1 -23095.601,E2 -23095.601} C_VEL
LIN {X 0,Y 188.017,Z 198.724,A -85,B 0,C 180,E1 -23096.435,E2 -23096.435} C_VEL
LIN {X 0,Y 189.918,Z 214.181,A -85,B 0,C 180,E1 -23097.493,E2 -23097.493} C_VEL
LIN {X 0,Y 188.663,Z 242.054,A -85,B 0,C 180,E1 -23098.566,E2 -23098.566} C_VEL
LIN {X 0,Y 187.474,Z 253.095,A -85,B 0,C 180,E1 -23099.285,E2 -23099.285} C_VEL
LIN {X 0,Y 185.623,Z 264.701,A -85,B 0,C 180,E1 -23100.515,E2 -23100.515} C_VEL
LIN {X 0,Y 183.702,Z 274.003,A -85,B 0,C 180,E1 -23101.875,E2 -23101.875} C_VEL
LIN {X 0,Y 181.867,Z 281.647,A -85,B 0,C 180,E1 -23103.306,E2 -23103.306} C_VEL
LIN {X 0,Y 179.669,Z 289.489,A -85,B 0,C 180,E1 -23105.135,E2 -23105.135} C_VEL
LIN {X 0,Y 177.433,Z 296.826,A -85,B 0,C 180,E1 -23107.283,E2 -23107.283} C_VEL
LIN {X 0,Y 174.954,Z 304.268,A -85,B 0,C 180,E1 -23110.035,E2 -23110.035} C_VEL
LIN {X 0,Y 174.023,Z 306.867,A -85,B 0,C 180,E1 -23111.247,E2 -23111.247} C_VEL
LIN {X 0,Y 172.309,Z 310.093,A -85,B 0,C 180,E1 -23112.802,E2 -23112.802} C_VEL
LIN {X 0,Y 167.999,Z 314.664,A -85,B 0,C 180,E1 -23115.387,E2 -23115.387} C_VEL
LIN {X 0,Y 163.937,Z 318.324,A -85,B 0,C 180,E1 -23118.246,E2 -23118.246} C_VEL
LIN {X 0,Y 162.662,Z 319.988,A -85,B 0,C 180,E1 -23120.186,E2 -23120.186} C_VEL
LIN {X 0,Y 162.149,Z 321.632,A -85,B 0,C 180,E1 -23122.529,E2 -23122.529} C_VEL
LIN {X 0,Y 161.858,Z 322.878,A -85,B 0,C 180,E1 -23125.019,E2 -23125.019} C_VEL
LIN {X 0,Y 161.763,Z 323.688,A -85,B 0,C 180,E1 -23127.791,E2 -23127.791} C_VEL
LIN {X 0,Y 161.801,Z 323.944,A -85,B 0,C 180,E1 -23130.001,E2 -23130.001} C_VEL
LIN {X 0,Y 161.759,Z 323.641,A -85,B 0,C 180,E1 -23132.491,E2 -23132.491} C_VEL
LIN {X 0,Y 161.858,Z 322.845,A -85,B 0,C 180,E1 -23134.983,E2 -23134.983} C_VEL
LIN {X 0,Y 162.145,Z 321.577,A -85,B 0,C 180,E1 -23137.472,E2 -23137.472} C_VEL
LIN {X 0,Y 163.013,Z 318.657,A -85,B 0,C 180,E1 -23141.187,E2 -23141.187} C_VEL
LIN {X 0,Y 163.892,Z 315.996,A -85,B 0,C 180,E1 -23143.642,E2 -23143.642} C_VEL
LIN {X 0,Y 165.791,Z 310.802,A -85,B 0,C 180,E1 -23147.262,E2 -23147.262} C_VEL
LIN {X 0,Y 168.288,Z 303.952,A -85,B 0,C 180,E1 -23150.792,E2 -23150.792} C_VEL
LIN {X 0,Y 170.915,Z 296.473,A -85,B 0,C 180,E1 -23153.636,E2 -23153.636} C_VEL
LIN {X 0,Y 173.228,Z 289.094,A -85,B 0,C 180,E1 -23155.858,E2 -23155.858} C_VEL
LIN {X 0,Y 175.55,Z 281.192,A -85,B 0,C 180,E1 -23157.736,E2 -23157.736} C_VEL
LIN {X 0,Y 177.812,Z 272.258,A -85,B 0,C 180,E1 -23159.408,E2 -23159.408} C_VEL
LIN {X 0,Y 179.998,Z 260.992,A -85,B 0,C 180,E1 -23160.992,E2 -23160.992} C_VEL
LIN {X 0,Y 181.617,Z 250.424,A -85,B 0,C 180,E1 -23161.983,E2 -23161.983} C_VEL
LIN {X 0,Y 182.636,Z 240.528,A -85,B 0,C 180,E1 -23162.598,E2 -23162.598} C_VEL
LIN {X 0,Y 183.768,Z 214.248,A -85,B 0,C 180,E1 -23163.64,E2 -23163.64} C_VEL
LIN {X 0,Y 181.908,Z 200.393,A -85,B 0,C 180,E1 -23164.677,E2 -23164.677} C_VEL
LIN {X 0,Y 177.571,Z 189.498,A -85,B 0,C 180,E1 -23166.177,E2 -23166.177} C_VEL
LIN {X 0,Y 171.396,Z 176.419,A -85,B 0,C 180,E1 -23168.373,E2 -23168.373} C_VEL
LIN {X 0,Y 166.494,Z 167.539,A -85,B 0,C 180,E1 -23170.203,E2 -23170.203} C_VEL
LIN {X 0,Y 164.486,Z 163.732,A -85,B 0,C 180,E1 -23171.145,E2 -23171.145} C_VEL
LIN {X 0,Y 164.342,Z 163.062,A -85,B 0,C 180,E1 -23171.552,E2 -23171.552} C_VEL
LIN {X 0,Y 164.28,Z 162.768,A -85,B 0,C 180,E1 -23176.659,E2 -23176.659} C_VEL
LIN {X 0,Y 164.296,Z 162.812,A -85,B 0,C 180,E1 -23180.352,E2 -23180.352} C_VEL
LIN {X 0,Y 164.331,Z 162.811,A -85,B 0,C 180,E1 -23186.222,E2 -23186.222} C_VEL
LIN {X 0,Y 164.407,Z 162.817,A -85,B 0,C 180,E1 -23189.138,E2 -23189.138} C_VEL
LIN {X 0,Y 164.418,Z 162.809,A -85,B 0,C 180,E1 -23194.695,E2 -23194.695} C_VEL
LIN {X 0,Y 164.487,Z 162.778,A -85,B 0,C 180,E1 -23200.051,E2 -23200.051} C_VEL
LIN {X 0,Y 164.543,Z 162.801,A -85,B 0,C 180,E1 -23205.151,E2 -23205.151} C_VEL
LIN {X 0,Y 164.771,Z 162.738,A -85,B 0,C 180,E1 -23210.177,E2 -23210.177} C_VEL
LIN {X 0,Y 164.836,Z 162.756,A -85,B 0,C 180,E1 -23212.652,E2 -23212.652} C_VEL
LIN {X 0,Y 165.05,Z 162.709,A -85,B 0,C 180,E1 -23217.56,E2 -23217.56} C_VEL
LIN {X 0,Y 165.296,Z 162.672,A -85,B 0,C 180,E1 -23220,E2 -23220} C_VEL
LIN {X 0,Y 164.775,Z 162.771,A -85,B 0,C 180,E1 -23224.894,E2 -23224.894} C_VEL
LIN {X 0,Y 164.849,Z 162.735,A -85,B 0,C 180,E1 -23227.348,E2 -23227.348} C_VEL
LIN {X 0,Y 164.753,Z 162.754,A -85,B 0,C 180,E1 -23231.146,E2 -23231.146} C_VEL
LIN {X 0,Y 164.507,Z 162.775,A -85,B 0,C 180,E1 -23237.401,E2 -23237.401} C_VEL
LIN {X 0,Y 164.476,Z 162.786,A -85,B 0,C 180,E1 -23239.989,E2 -23239.989} C_VEL
LIN {X 0,Y 164.396,Z 162.792,A -85,B 0,C 180,E1 -23246.134,E2 -23246.134} C_VEL
LIN {X 0,Y 164.391,Z 162.818,A -85,B 0,C 180,E1 -23251.236,E2 -23251.236} C_VEL
LIN {X 0,Y 164.297,Z 162.832,A -85,B 0,C 180,E1 -23256.789,E2 -23256.789} C_VEL
LIN {X 0,Y 164.294,Z 162.816,A -85,B 0,C 180,E1 -23259.916,E2 -23259.916} C_VEL
LIN {X 0,Y 164.281,Z 162.833,A -85,B 0,C 180,E1 -23263.342,E2 -23263.342} C_VEL
LIN {X 0,Y 164.337,Z 162.924,A -85,B 0,C 180,E1 -23268.682,E2 -23268.682} C_VEL
LIN {X 0,Y 164.476,Z 163.712,A -85,B 0,C 180,E1 -23269.21,E2 -23269.21} C_VEL
LIN {X 0,Y 165.978,Z 166.54,A -85,B 0,C 180,E1 -23269.891,E2 -23269.891} C_VEL
LIN {X 0,Y 167.333,Z 168.354,A -85,B 0,C 180,E1 -23270.383,E2 -23270.383} C_VEL
LIN {X 0,Y 174.028,Z 179.2,A -85,B 0,C 180,E1 -23272.747,E2 -23272.747} C_VEL
LIN {X 0,Y 178.026,Z 186.736,A -85,B 0,C 180,E1 -23274.094,E2 -23274.094} C_VEL
LIN {X 0,Y 183.15,Z 199.242,A -85,B 0,C 180,E1 -23275.836,E2 -23275.836} C_VEL
LIN {X 0,Y 184.436,Z 202.923,A -85,B 0,C 180,E1 -23276.278,E2 -23276.278} C_VEL
LIN {X 0,Y 182.763,Z 235.739,A -85,B 0,C 180,E1 -23277.522,E2 -23277.522} C_VEL
LIN {X 0,Y 181.754,Z 246.223,A -85,B 0,C 180,E1 -23278.224,E2 -23278.224} C_VEL
LIN {X 0,Y 180.001,Z 258.212,A -85,B 0,C 180,E1 -23279.497,E2 -23279.497} C_VEL
LIN {X 0,Y 178.244,Z 267.009,A -85,B 0,C 180,E1 -23280.794,E2 -23280.794} C_VEL
LIN {X 0,Y 176.244,Z 275.384,A -85,B 0,C 180,E1 -23282.382,E2 -23282.382} C_VEL
LIN {X 0,Y 173.937,Z 283.297,A -85,B 0,C 180,E1 -23284.255,E2 -23284.255} C_VEL
LIN {X 0,Y 171.607,Z 290.674,A -85,B 0,C 180,E1 -23286.465,E2 -23286.465} C_VEL
LIN {X 0,Y 169.064,Z 298.146,A -85,B 0,C 180,E1 -23289.307,E2 -23289.307} C_VEL
LIN {X 0,Y 166.478,Z 304.993,A -85,B 0,C 180,E1 -23292.811,E2 -23292.811} C_VEL
LIN {X 0,Y 164.533,Z 310.167,A -85,B 0,C 180,E1 -23296.412,E2 -23296.412} C_VEL
LIN {X 0,Y 163.555,Z 312.82,A -85,B 0,C 180,E1 -23298.85,E2 -23298.85} C_VEL
LIN {X 0,Y 162.554,Z 315.723,A -85,B 0,C 180,E1 -23302.547,E2 -23302.547} C_VEL
LIN {X 0,Y 161.966,Z 317.516,A -85,B 0,C 180,E1 -23306.392,E2 -23306.392} C_VEL
LIN {X 0,Y 161.841,Z 318.088,A -85,B 0,C 180,E1 -23309.999,E2 -23309.999} C_VEL
LIN {X 0,Y 161.938,Z 317.634,A -85,B 0,C 180,E1 -23313.45,E2 -23313.45} C_VEL
LIN {X 0,Y 162.485,Z 315.838,A -85,B 0,C 180,E1 -23317.455,E2 -23317.455} C_VEL
LIN {X 0,Y 163.548,Z 312.98,A -85,B 0,C 180,E1 -23321.149,E2 -23321.149} C_VEL
LIN {X 0,Y 164.502,Z 310.378,A -85,B 0,C 180,E1 -23323.59,E2 -23323.59} C_VEL
LIN {X 0,Y 166.45,Z 305.26,A -85,B 0,C 180,E1 -23327.19,E2 -23327.19} C_VEL
LIN {X 0,Y 168.554,Z 299.751,A -85,B 0,C 180,E1 -23330.12,E2 -23330.12} C_VEL
LIN {X 0,Y 171.013,Z 292.825,A -85,B 0,C 180,E1 -23332.98,E2 -23332.98} C_VEL
LIN {X 0,Y 173.602,Z 284.871,A -85,B 0,C 180,E1 -23335.476,E2 -23335.476} C_VEL
LIN {X 0,Y 175.861,Z 277.285,A -85,B 0,C 180,E1 -23337.359,E2 -23337.359} C_VEL
LIN {X 0,Y 177.835,Z 269.332,A -85,B 0,C 180,E1 -23338.954,E2 -23338.954} C_VEL
LIN {X 0,Y 179.616,Z 261.108,A -85,B 0,C 180,E1 -23340.249,E2 -23340.249} C_VEL
LIN {X 0,Y 181.024,Z 252.798,A -85,B 0,C 180,E1 -23341.277,E2 -23341.277} C_VEL
LIN {X 0,Y 182.17,Z 243.987,A -85,B 0,C 180,E1 -23342.091,E2 -23342.091} C_VEL
LIN {X 0,Y 182.954,Z 234.697,A -85,B 0,C 180,E1 -23342.684,E2 -23342.684} C_VEL
LIN {X 0,Y 184.511,Z 202.948,A -85,B 0,C 180,E1 -23343.884,E2 -23343.884} C_VEL
LIN {X 0,Y 180.316,Z 191.893,A -85,B 0,C 180,E1 -23345.315,E2 -23345.315} C_VEL
LIN {X 0,Y 175.972,Z 182.52,A -85,B 0,C 180,E1 -23346.795,E2 -23346.795} C_VEL
LIN {X 0,Y 169.274,Z 171.312,A -85,B 0,C 180,E1 -23349.115,E2 -23349.115} C_VEL
LIN {X 0,Y 167.015,Z 167.762,A -85,B 0,C 180,E1 -23349.946,E2 -23349.946} C_VEL
LIN {X 0,Y 164.915,Z 164.878,A -85,B 0,C 180,E1 -23350.728,E2 -23350.728} C_VEL
LIN {X 0,Y 164.372,Z 163.204,A -85,B 0,C 180,E1 -23351.216,E2 -23351.216} C_VEL
LIN {X 0,Y 164.291,Z 162.778,A -85,B 0,C 180,E1 -23352.253,E2 -23352.253} C_VEL
LIN {X 0,Y 164.292,Z 162.831,A -85,B 0,C 180,E1 -23356.808,E2 -23356.808} C_VEL
LIN {X 0,Y 164.295,Z 162.816,A -85,B 0,C 180,E1 -23360.351,E2 -23360.351} C_VEL
LIN {X 0,Y 164.329,Z 162.805,A -85,B 0,C 180,E1 -23366.221,E2 -23366.221} C_VEL
LIN {X 0,Y 164.405,Z 162.817,A -85,B 0,C 180,E1 -23369.137,E2 -23369.137} C_VEL
LIN {X 0,Y 164.416,Z 162.793,A -85,B 0,C 180,E1 -23374.694,E2 -23374.694} C_VEL
LIN {X 0,Y 164.484,Z 162.786,A -85,B 0,C 180,E1 -23380.051,E2 -23380.051} C_VEL
LIN {X 0,Y 164.553,Z 162.795,A -85,B 0,C 180,E1 -23385.152,E2 -23385.152} C_VEL
LIN {X 0,Y 164.797,Z 162.736,A -85,B 0,C 180,E1 -23390.178,E2 -23390.178} C_VEL
LIN {X 0,Y 164.846,Z 162.735,A -85,B 0,C 180,E1 -23392.651,E2 -23392.651} C_VEL
LIN {X 0,Y 165.05,Z 162.729,A -85,B 0,C 180,E1 -23397.559,E2 -23397.559} C_VEL
LIN {X 0,Y 165.295,Z 162.672,A -85,B 0,C 180,E1 -23400,E2 -23400} C_VEL
LIN {X 0,Y 164.774,Z 162.771,A -85,B 0,C 180,E1 -23404.893,E2 -23404.893} C_VEL
LIN {X 0,Y 164.854,Z 162.754,A -85,B 0,C 180,E1 -23407.348,E2 -23407.348} C_VEL
LIN {X 0,Y 164.743,Z 162.742,A -85,B 0,C 180,E1 -23411.135,E2 -23411.135} C_VEL
LIN {X 0,Y 164.504,Z 162.79,A -85,B 0,C 180,E1 -23417.401,E2 -23417.401} C_VEL
LIN {X 0,Y 164.472,Z 162.78,A -85,B 0,C 180,E1 -23419.989,E2 -23419.989} C_VEL
LIN {X 0,Y 164.392,Z 162.801,A -85,B 0,C 180,E1 -23426.134,E2 -23426.134} C_VEL
LIN {X 0,Y 164.387,Z 162.822,A -85,B 0,C 180,E1 -23431.236,E2 -23431.236} C_VEL
LIN {X 0,Y 164.293,Z 162.825,A -85,B 0,C 180,E1 -23436.789,E2 -23436.789} C_VEL
LIN {X 0,Y 164.289,Z 162.804,A -85,B 0,C 180,E1 -23439.916,E2 -23439.916} C_VEL
LIN {X 0,Y 164.278,Z 162.768,A -85,B 0,C 180,E1 -23443.342,E2 -23443.342} C_VEL
LIN {X 0,Y 164.34,Z 163.05,A -85,B 0,C 180,E1 -23448.324,E2 -23448.324} C_VEL
LIN {X 0,Y 164.659,Z 164.243,A -85,B 0,C 180,E1 -23448.902,E2 -23448.902} C_VEL
LIN {X 0,Y 168.084,Z 170.332,A -85,B 0,C 180,E1 -23450.29,E2 -23450.29} C_VEL
LIN {X 0,Y 173.441,Z 180.471,A -85,B 0,C 180,E1 -23452.261,E2 -23452.261} C_VEL
LIN {X 0,Y 179.914,Z 194.889,A -85,B 0,C 180,E1 -23454.528,E2 -23454.528} C_VEL
LIN {X 0,Y 182.375,Z 201.826,A -85,B 0,C 180,E1 -23455.4,E2 -23455.4} C_VEL
LIN {X 0,Y 183.94,Z 215.329,A -85,B 0,C 180,E1 -23456.356,E2 -23456.356} C_VEL
LIN {X 0,Y 182.634,Z 241.941,A -85,B 0,C 180,E1 -23457.403,E2 -23457.403} C_VEL
LIN {X 0,Y 181.413,Z 252.976,A -85,B 0,C 180,E1 -23458.141,E2 -23458.141} C_VEL
LIN {X 0,Y 179.488,Z 264.578,A -85,B 0,C 180,E1 -23459.402,E2 -23459.402} C_VEL
LIN {X 0,Y 177.704,Z 272.899,A -85,B 0,C 180,E1 -23460.625,E2 -23460.625} C_VEL
LIN {X 0,Y 175.565,Z 281.523,A -85,B 0,C 180,E1 -23462.267,E2 -23462.267} C_VEL
LIN {X 0,Y 173.234,Z 289.364,A -85,B 0,C 180,E1 -23464.144,E2 -23464.144} C_VEL
LIN {X 0,Y 170.906,Z 296.7,A -85,B 0,C 180,E1 -23466.364,E2 -23466.364} C_VEL
LIN {X 0,Y 168.299,Z 304.142,A -85,B 0,C 180,E1 -23469.21,E2 -23469.21} C_VEL
LIN {X 0,Y 166.191,Z 309.975,A -85,B 0,C 180,E1 -23472.147,E2 -23472.147} C_VEL
LIN {X 0,Y 164.475,Z 314.576,A -85,B 0,C 180,E1 -23475.145,E2 -23475.145} C_VEL
LIN {X 0,Y 163.457,Z 317.568,A -85,B 0,C 180,E1 -23477.586,E2 -23477.586} C_VEL
LIN {X 0,Y 162.662,Z 319.988,A -85,B 0,C 180,E1 -23480.186,E2 -23480.186} C_VEL
LIN {X 0,Y 161.554,Z 321.437,A -85,B 0,C 180,E1 -23482.185,E2 -23482.185} C_VEL
LIN {X 0,Y 159.71,Z 322.537,A -85,B 0,C 180,E1 -23484.166,E2 -23484.166} C_VEL
LIN {X 0,Y 155.808,Z 323.69,A -85,B 0,C 180,E1 -23488.249,E2 -23488.249} C_VEL
LIN {X 0,Y 154.747,Z 323.786,A -85,B 0,C 180,E1 -23490.412,E2 -23490.412} C_VEL
LIN {X 0,Y 154.657,Z 323.691,A -85,B 0,C 180,E1 -23491.146,E2 -23491.146} C_VEL
LIN {X 0,Y 154.771,Z 322.716,A -85,B 0,C 180,E1 -23495.211,E2 -23495.211} C_VEL
LIN {X 0,Y 155.086,Z 321.448,A -85,B 0,C 180,E1 -23497.814,E2 -23497.814} C_VEL
LIN {X 0,Y 156.028,Z 318.528,A -85,B 0,C 180,E1 -23501.695,E2 -23501.695} C_VEL
LIN {X 0,Y 156.993,Z 315.867,A -85,B 0,C 180,E1 -23504.254,E2 -23504.254} C_VEL
LIN {X 0,Y 159.004,Z 310.672,A -85,B 0,C 180,E1 -23508.024,E2 -23508.024} C_VEL
LIN {X 0,Y 161.676,Z 303.822,A -85,B 0,C 180,E1 -23511.685,E2 -23511.685} C_VEL
LIN {X 0,Y 164.437,Z 296.342,A -85,B 0,C 180,E1 -23514.628,E2 -23514.628} C_VEL
LIN {X 0,Y 166.864,Z 288.963,A -85,B 0,C 180,E1 -23516.922,E2 -23516.922} C_VEL
LIN {X 0,Y 169.308,Z 281.06,A -85,B 0,C 180,E1 -23518.853,E2 -23518.853} C_VEL
LIN {X 0,Y 171.867,Z 271.237,A -85,B 0,C 180,E1 -23520.733,E2 -23520.733} C_VEL
LIN {X 0,Y 174.144,Z 259.799,A -85,B 0,C 180,E1 -23522.305,E2 -23522.305} C_VEL
LIN {X 0,Y 175.685,Z 250.061,A -85,B 0,C 180,E1 -23523.222,E2 -23523.222} C_VEL
LIN {X 0,Y 176.687,Z 240.384,A -85,B 0,C 180,E1 -23523.84,E2 -23523.84} C_VEL
LIN {X 0,Y 177.909,Z 215.46,A -85,B 0,C 180,E1 -23524.84,E2 -23524.84} C_VEL
LIN {X 0,Y 176.304,Z 203.045,A -85,B 0,C 180,E1 -23525.809,E2 -23525.809} C_VEL
LIN {X 0,Y 172.706,Z 193.802,A -85,B 0,C 180,E1 -23527.14,E2 -23527.14} C_VEL
LIN {X 0,Y 166.801,Z 180.906,A -85,B 0,C 180,E1 -23529.383,E2 -23529.383} C_VEL
LIN {X 0,Y 161.82,Z 171.817,A -85,B 0,C 180,E1 -23531.361,E2 -23531.361} C_VEL
LIN {X 0,Y 159.602,Z 168.161,A -85,B 0,C 180,E1 -23532.279,E2 -23532.279} C_VEL
LIN {X 0,Y 157.795,Z 165.693,A -85,B 0,C 180,E1 -23533.036,E2 -23533.036} C_VEL
LIN {X 0,Y 157.387,Z 164.41,A -85,B 0,C 180,E1 -23533.389,E2 -23533.389} C_VEL
LIN {X 0,Y 157.215,Z 163.744,A -85,B 0,C 180,E1 -23534.085,E2 -23534.085} C_VEL
LIN {X 0,Y 157.199,Z 163.674,A -85,B 0,C 180,E1 -23539.468,E2 -23539.468} C_VEL
LIN {X 0,Y 157.28,Z 163.686,A -85,B 0,C 180,E1 -23544.486,E2 -23544.486} C_VEL
LIN {X 0,Y 157.303,Z 163.704,A -85,B 0,C 180,E1 -23548.092,E2 -23548.092} C_VEL
LIN {X 0,Y 157.323,Z 163.678,A -85,B 0,C 180,E1 -23553.467,E2 -23553.467} C_VEL
LIN {X 0,Y 157.395,Z 163.661,A -85,B 0,C 180,E1 -23559.668,E2 -23559.668} C_VEL
LIN {X 0,Y 157.472,Z 163.682,A -85,B 0,C 180,E1 -23564.468,E2 -23564.468} C_VEL
LIN {X 0,Y 157.692,Z 163.618,A -85,B 0,C 180,E1 -23569.731,E2 -23569.731} C_VEL
LIN {X 0,Y 157.773,Z 163.631,A -85,B 0,C 180,E1 -23572.321,E2 -23572.321} C_VEL
LIN {X 0,Y 158.258,Z 163.547,A -85,B 0,C 180,E1 -23580,E2 -23580} C_VEL
LIN {X 0,Y 157.787,Z 163.61,A -85,B 0,C 180,E1 -23587.679,E2 -23587.679} C_VEL
LIN {X 0,Y 157.683,Z 163.635,A -85,B 0,C 180,E1 -23591.317,E2 -23591.317} C_VEL
LIN {X 0,Y 157.481,Z 163.669,A -85,B 0,C 180,E1 -23595.532,E2 -23595.532} C_VEL
LIN {X 0,Y 157.372,Z 163.681,A -85,B 0,C 180,E1 -23600.933,E2 -23600.933} C_VEL
LIN {X 0,Y 157.317,Z 163.673,A -85,B 0,C 180,E1 -23606.684,E2 -23606.684} C_VEL
LIN {X 0,Y 157.284,Z 163.688,A -85,B 0,C 180,E1 -23612.426,E2 -23612.426} C_VEL
LIN {X 0,Y 157.27,Z 163.704,A -85,B 0,C 180,E1 -23616.449,E2 -23616.449} C_VEL
LIN {X 0,Y 157.213,Z 163.71,A -85,B 0,C 180,E1 -23622.11,E2 -23622.11} C_VEL
LIN {X 0,Y 157.234,Z 163.797,A -85,B 0,C 180,E1 -23626.411,E2 -23626.411} C_VEL
LIN {X 0,Y 157.444,Z 164.665,A -85,B 0,C 180,E1 -23627.029,E2 -23627.029} C_VEL
LIN {X 0,Y 158.943,Z 167.474,A -85,B 0,C 180,E1 -23627.764,E2 -23627.764} C_VEL
LIN {X 0,Y 160.36,Z 169.218,A -85,B 0,C 180,E1 -23628.327,E2 -23628.327} C_VEL
LIN {X 0,Y 167.433,Z 180.375,A -85,B 0,C 180,E1 -23631.065,E2 -23631.065} C_VEL
LIN {X 0,Y 172.675,Z 189.864,A -85,B 0,C 180,E1 -23632.951,E2 -23632.951} C_VEL
LIN {X 0,Y 177.871,Z 202.767,A -85,B 0,C 180,E1 -23634.839,E2 -23634.839} C_VEL
LIN {X 0,Y 178.523,Z 205.359,A -85,B 0,C 180,E1 -23635.112,E2 -23635.112} C_VEL
LIN {X 0,Y 176.816,Z 235.538,A -85,B 0,C 180,E1 -23636.264,E2 -23636.264} C_VEL
LIN {X 0,Y 175.897,Z 245.475,A -85,B 0,C 180,E1 -23636.944,E2 -23636.944} C_VEL
LIN {X 0,Y 174.307,Z 256.401,A -85,B 0,C 180,E1 -23638.053,E2 -23638.053} C_VEL
LIN {X 0,Y 172.098,Z 267.142,A -85,B 0,C 180,E1 -23639.644,E2 -23639.644} C_VEL
LIN {X 0,Y 169.999,Z 275.517,A -85,B 0,C 180,E1 -23641.275,E2 -23641.275} C_VEL
LIN {X 0,Y 167.582,Z 283.428,A -85,B 0,C 180,E1 -23643.202,E2 -23643.202} C_VEL
LIN {X 0,Y 165.129,Z 290.805,A -85,B 0,C 180,E1 -23645.482,E2 -23645.482} C_VEL
LIN {X 0,Y 162.446,Z 298.277,A -85,B 0,C 180,E1 -23648.423,E2 -23648.423} C_VEL
LIN {X 0,Y 159.707,Z 305.123,A -85,B 0,C 180,E1 -23652.058,E2 -23652.058} C_VEL
LIN {X 0,Y 157.646,Z 310.297,A -85,B 0,C 180,E1 -23655.806,E2 -23655.806} C_VEL
LIN {X 0,Y 156.583,Z 312.949,A -85,B 0,C 180,E1 -23658.347,E2 -23658.347} C_VEL
LIN {X 0,Y 155.515,Z 315.853,A -85,B 0,C 180,E1 -23662.207,E2 -23662.207} C_VEL
LIN {X 0,Y 155.057,Z 317.118,A -85,B 0,C 180,E1 -23664.798,E2 -23664.798} C_VEL
LIN {X 0,Y 154.777,Z 317.914,A -85,B 0,C 180,E1 -23667.397,E2 -23667.397} C_VEL
LIN {X 0,Y 154.745,Z 318.216,A -85,B 0,C 180,E1 -23669.999,E2 -23669.999} C_VEL
LIN {X 0,Y 154.776,Z 317.936,A -85,B 0,C 180,E1 -23672.602,E2 -23672.602} C_VEL
LIN {X 0,Y 155.054,Z 317.184,A -85,B 0,C 180,E1 -23675.2,E2 -23675.2} C_VEL
LIN {X 0,Y 155.443,Z 315.966,A -85,B 0,C 180,E1 -23677.795,E2 -23677.795} C_VEL
LIN {X 0,Y 156.576,Z 313.108,A -85,B 0,C 180,E1 -23681.652,E2 -23681.652} C_VEL
LIN {X 0,Y 157.616,Z 310.505,A -85,B 0,C 180,E1 -23684.195,E2 -23684.195} C_VEL
LIN {X 0,Y 159.674,Z 305.387,A -85,B 0,C 180,E1 -23687.944,E2 -23687.944} C_VEL
LIN {X 0,Y 161.904,Z 299.878,A -85,B 0,C 180,E1 -23690.984,E2 -23690.984} C_VEL
LIN {X 0,Y 164.506,Z 292.951,A -85,B 0,C 180,E1 -23693.944,E2 -23693.944} C_VEL
LIN {X 0,Y 167.224,Z 284.996,A -85,B 0,C 180,E1 -23696.521,E2 -23696.521} C_VEL
LIN {X 0,Y 169.606,Z 277.409,A -85,B 0,C 180,E1 -23698.458,E2 -23698.458} C_VEL
LIN {X 0,Y 171.669,Z 269.455,A -85,B 0,C 180,E1 -23700.099,E2 -23700.099} C_VEL
LIN {X 0,Y 173.539,Z 261.23,A -85,B 0,C 180,E1 -23701.426,E2 -23701.426} C_VEL
LIN {X 0,Y 174.906,Z 253.588,A -85,B 0,C 180,E1 -23702.408,E2 -23702.408} C_VEL
LIN {X 0,Y 176.246,Z 243.827,A -85,B 0,C 180,E1 -23703.335,E2 -23703.335} C_VEL
LIN {X 0,Y 177.054,Z 234.602,A -85,B 0,C 180,E1 -23703.931,E2 -23703.931} C_VEL
LIN {X 0,Y 178.54,Z 204.527,A -85,B 0,C 180,E1 -23705.11,E2 -23705.11} C_VEL
LIN {X 0,Y 173.7,Z 192.081,A -85,B 0,C 180,E1 -23706.873,E2 -23706.873} C_VEL
LIN {X 0,Y 170.242,Z 185.192,A -85,B 0,C 180,E1 -23708.116,E2 -23708.116} C_VEL
LIN {X 0,Y 164.562,Z 175.761,A -85,B 0,C 180,E1 -23710.217,E2 -23710.217} C_VEL
LIN {X 0,Y 161.693,Z 171.454,A -85,B 0,C 180,E1 -23711.335,E2 -23711.335} C_VEL
LIN {X 0,Y 159.637,Z 168.151,A -85,B 0,C 180,E1 -23712.186,E2 -23712.186} C_VEL
LIN {X 0,Y 157.855,Z 165.717,A -85,B 0,C 180,E1 -23712.931,E2 -23712.931} C_VEL
LIN {X 0,Y 157.345,Z 164.25,A -85,B 0,C 180,E1 -23713.373,E2 -23713.373} C_VEL
LIN {X 0,Y 157.18,Z 163.699,A -85,B 0,C 180,E1 -23714.323,E2 -23714.323} C_VEL
LIN {X 0,Y 157.205,Z 163.699,A -85,B 0,C 180,E1 -23719.463,E2 -23719.463} C_VEL
LIN {X 0,Y 157.278,Z 163.693,A -85,B 0,C 180,E1 -23724.485,E2 -23724.485} C_VEL
LIN {X 0,Y 157.301,Z 163.69,A -85,B 0,C 180,E1 -23728.09,E2 -23728.09} C_VEL
LIN {X 0,Y 157.321,Z 163.672,A -85,B 0,C 180,E1 -23733.466,E2 -23733.466} C_VEL
LIN {X 0,Y 157.393,Z 163.672,A -85,B 0,C 180,E1 -23739.667,E2 -23739.667} C_VEL
LIN {X 0,Y 157.477,Z 163.667,A -85,B 0,C 180,E1 -23744.468,E2 -23744.468} C_VEL
LIN {X 0,Y 157.725,Z 163.619,A -85,B 0,C 180,E1 -23749.733,E2 -23749.733} C_VEL
LIN {X 0,Y 157.784,Z 163.61,A -85,B 0,C 180,E1 -23752.321,E2 -23752.321} C_VEL
LIN {X 0,Y 158.257,Z 163.548,A -85,B 0,C 180,E1 -23760,E2 -23760} C_VEL
LIN {X 0,Y 157.81,Z 163.626,A -85,B 0,C 180,E1 -23767.678,E2 -23767.678} C_VEL
LIN {X 0,Y 157.675,Z 163.622,A -85,B 0,C 180,E1 -23771.308,E2 -23771.308} C_VEL
LIN {X 0,Y 157.477,Z 163.681,A -85,B 0,C 180,E1 -23775.531,E2 -23775.531} C_VEL
LIN {X 0,Y 157.369,Z 163.669,A -85,B 0,C 180,E1 -23780.933,E2 -23780.933} C_VEL
LIN {X 0,Y 157.313,Z 163.678,A -85,B 0,C 180,E1 -23786.684,E2 -23786.684} C_VEL
LIN {X 0,Y 157.28,Z 163.701,A -85,B 0,C 180,E1 -23792.426,E2 -23792.426} C_VEL
LIN {X 0,Y 157.266,Z 163.695,A -85,B 0,C 180,E1 -23796.45,E2 -23796.45} C_VEL
LIN {X 0,Y 157.19,Z 163.654,A -85,B 0,C 180,E1 -23802.117,E2 -23802.117} C_VEL
LIN {X 0,Y 157.25,Z 163.947,A -85,B 0,C 180,E1 -23806.155,E2 -23806.155} C_VEL
LIN {X 0,Y 157.539,Z 165.058,A -85,B 0,C 180,E1 -23806.68,E2 -23806.68} C_VEL
LIN {X 0,Y 159.221,Z 167.826,A -85,B 0,C 180,E1 -23807.448,E2 -23807.448} C_VEL
LIN {X 0,Y 160.287,Z 169.143,A -85,B 0,C 180,E1 -23807.874,E2 -23807.874} C_VEL
LIN {X 0,Y 165.215,Z 177.766,A -85,B 0,C 180,E1 -23809.877,E2 -23809.877} C_VEL
LIN {X 0,Y 171.423,Z 190.77,A -85,B 0,C 180,E1 -23812.274,E2 -23812.274} C_VEL
LIN {X 0,Y 175.992,Z 201.937,A -85,B 0,C 180,E1 -23813.965,E2 -23813.965} C_VEL
LIN {X 0,Y 176.829,Z 205.19,A -85,B 0,C 180,E1 -23814.321,E2 -23814.321} C_VEL
LIN {X 0,Y 178.032,Z 216.328,A -85,B 0,C 180,E1 -23815.135,E2 -23815.135} C_VEL
LIN {X 0,Y 176.692,Z 241.829,A -85,B 0,C 180,E1 -23816.162,E2 -23816.162} C_VEL
LIN {X 0,Y 175.439,Z 252.882,A -85,B 0,C 180,E1 -23816.923,E2 -23816.923} C_VEL
LIN {X 0,Y 173.41,Z 264.456,A -85,B 0,C 180,E1 -23818.207,E2 -23818.207} C_VEL
LIN {X 0,Y 171.558,Z 272.776,A -85,B 0,C 180,E1 -23819.462,E2 -23819.462} C_VEL
LIN {X 0,Y 169.321,Z 281.398,A -85,B 0,C 180,E1 -23821.151,E2 -23821.151} C_VEL
LIN {X 0,Y 166.876,Z 289.238,A -85,B 0,C 180,E1 -23823.081,E2 -23823.081} C_VEL
LIN {X 0,Y 164.425,Z 296.574,A -85,B 0,C 180,E1 -23825.372,E2 -23825.372} C_VEL
LIN {X 0,Y 161.684,Z 304.015,A -85,B 0,C 180,E1 -23828.318,E2 -23828.318} C_VEL
LIN {X 0,Y 159.413,Z 309.848,A -85,B 0,C 180,E1 -23831.36,E2 -23831.36} C_VEL
LIN {X 0,Y 157.612,Z 314.448,A -85,B 0,C 180,E1 -23834.483,E2 -23834.483} C_VEL
LIN {X 0,Y 156.527,Z 317.441,A -85,B 0,C 180,E1 -23837.027,E2 -23837.027} C_VEL
LIN {X 0,Y 155.599,Z 319.989,A -85,B 0,C 180,E1 -23839.932,E2 -23839.932} C_VEL
LIN {X 0,Y 155.094,Z 321.504,A -85,B 0,C 180,E1 -23842.187,E2 -23842.187} C_VEL
LIN {X 0,Y 154.77,Z 322.75,A -85,B 0,C 180,E1 -23844.79,E2 -23844.79} C_VEL
LIN {X 0,Y 154.652,Z 323.692,A -85,B 0,C 180,E1 -23848.751,E2 -23848.751} C_VEL
LIN {X 0,Y 154.657,Z 323.691,A -85,B 0,C 180,E1 -23851.146,E2 -23851.146} C_VEL
LIN {X 0,Y 154.008,Z 323.388,A -85,B 0,C 180,E1 -23853.318,E2 -23853.318} C_VEL
LIN {X 0,Y 151.422,Z 322.053,A -85,B 0,C 180,E1 -23856.875,E2 -23856.875} C_VEL
LIN {X 0,Y 149.223,Z 319.869,A -85,B 0,C 180,E1 -23860.489,E2 -23860.489} C_VEL
LIN {X 0,Y 149.208,Z 318.028,A -85,B 0,C 180,E1 -23862.673,E2 -23862.673} C_VEL
LIN {X 0,Y 150.77,Z 314.214,A -85,B 0,C 180,E1 -23866.242,E2 -23866.242} C_VEL
LIN {X 0,Y 153.12,Z 308.484,A -85,B 0,C 180,E1 -23870.136,E2 -23870.136} C_VEL
LIN {X 0,Y 155.644,Z 302.274,A -85,B 0,C 180,E1 -23873.273,E2 -23873.273} C_VEL
LIN {X 0,Y 158.01,Z 296.211,A -85,B 0,C 180,E1 -23875.701,E2 -23875.701} C_VEL
LIN {X 0,Y 160.568,Z 288.831,A -85,B 0,C 180,E1 -23878.069,E2 -23878.069} C_VEL
LIN {X 0,Y 163.135,Z 280.928,A -85,B 0,C 180,E1 -23880.055,E2 -23880.055} C_VEL
LIN {X 0,Y 165.617,Z 271.845,A -85,B 0,C 180,E1 -23881.85,E2 -23881.85} C_VEL
LIN {X 0,Y 167.958,Z 260.983,A -85,B 0,C 180,E1 -23883.453,E2 -23883.453} C_VEL
LIN {X 0,Y 169.705,Z 250.705,A -85,B 0,C 180,E1 -23884.471,E2 -23884.471} C_VEL
LIN {X 0,Y 170.764,Z 241.42,A -85,B 0,C 180,E1 -23885.101,E2 -23885.101} C_VEL
LIN {X 0,Y 172.033,Z 216.004,A -85,B 0,C 180,E1 -23886.178,E2 -23886.178} C_VEL
LIN {X 0,Y 170.652,Z 205.287,A -85,B 0,C 180,E1 -23887.067,E2 -23887.067} C_VEL
LIN {X 0,Y 166.699,Z 195.253,A -85,B 0,C 180,E1 -23888.633,E2 -23888.633} C_VEL
LIN {X 0,Y 160.978,Z 182.948,A -85,B 0,C 180,E1 -23890.978,E2 -23890.978} C_VEL
LIN {X 0,Y 156.644,Z 175.055,A -85,B 0,C 180,E1 -23892.843,E2 -23892.843} C_VEL
LIN {X 0,Y 153.296,Z 169.898,A -85,B 0,C 180,E1 -23894.337,E2 -23894.337} C_VEL
LIN {X 0,Y 150.924,Z 167.037,A -85,B 0,C 180,E1 -23895.409,E2 -23895.409} C_VEL
LIN {X 0,Y 150.242,Z 165.203,A -85,B 0,C 180,E1 -23895.97,E2 -23895.97} C_VEL
LIN {X 0,Y 150.121,Z 164.609,A -85,B 0,C 180,E1 -23896.661,E2 -23896.661} C_VEL
LIN {X 0,Y 150.178,Z 164.588,A -85,B 0,C 180,E1 -23902.529,E2 -23902.529} C_VEL
LIN {X 0,Y 150.221,Z 164.577,A -85,B 0,C 180,E1 -23907.365,E2 -23907.365} C_VEL
LIN {X 0,Y 150.246,Z 164.554,A -85,B 0,C 180,E1 -23912.718,E2 -23912.718} C_VEL
LIN {X 0,Y 150.353,Z 164.539,A -85,B 0,C 180,E1 -23919.208,E2 -23919.208} C_VEL
LIN {X 0,Y 150.379,Z 164.56,A -85,B 0,C 180,E1 -23923.716,E2 -23923.716} C_VEL
LIN {X 0,Y 150.614,Z 164.498,A -85,B 0,C 180,E1 -23929.243,E2 -23929.243} C_VEL
LIN {X 0,Y 150.709,Z 164.503,A -85,B 0,C 180,E1 -23931.958,E2 -23931.958} C_VEL
LIN {X 0,Y 151.219,Z 164.423,A -85,B 0,C 180,E1 -23940,E2 -23940} C_VEL
LIN {X 0,Y 150.727,Z 164.486,A -85,B 0,C 180,E1 -23948.041,E2 -23948.041} C_VEL
LIN {X 0,Y 150.614,Z 164.516,A -85,B 0,C 180,E1 -23951.501,E2 -23951.501} C_VEL
LIN {X 0,Y 150.384,Z 164.54,A -85,B 0,C 180,E1 -23956.284,E2 -23956.284} C_VEL
LIN {X 0,Y 150.353,Z 164.552,A -85,B 0,C 180,E1 -23960.792,E2 -23960.792} C_VEL
LIN {X 0,Y 150.247,Z 164.554,A -85,B 0,C 180,E1 -23967.283,E2 -23967.283} C_VEL
LIN {X 0,Y 150.222,Z 164.565,A -85,B 0,C 180,E1 -23972.635,E2 -23972.635} C_VEL
LIN {X 0,Y 150.175,Z 164.591,A -85,B 0,C 180,E1 -23977.473,E2 -23977.473} C_VEL
LIN {X 0,Y 150.14,Z 164.598,A -85,B 0,C 180,E1 -23982.922,E2 -23982.922} C_VEL
LIN {X 0,Y 150.198,Z 164.953,A -85,B 0,C 180,E1 -23984.154,E2 -23984.154} C_VEL
LIN {X 0,Y 150.606,Z 166.372,A -85,B 0,C 180,E1 -23984.71,E2 -23984.71} C_VEL
LIN {X 0,Y 152.329,Z 168.863,A -85,B 0,C 180,E1 -23985.54,E2 -23985.54} C_VEL
LIN {X 0,Y 153.42,Z 170.113,A -85,B 0,C 180,E1 -23986.021,E2 -23986.021} C_VEL
LIN {X 0,Y 155.728,Z 173.544,A -85,B 0,C 180,E1 -23987.052,E2 -23987.052} C_VEL
LIN {X 0,Y 162.674,Z 184.481,A -85,B 0,C 180,E1 -23989.923,E2 -23989.923} C_VEL
LIN {X 0,Y 167.767,Z 193.944,A -85,B 0,C 180,E1 -23991.886,E2 -23991.886} C_VEL
LIN {X 0,Y 172.576,Z 206.113,A -85,B 0,C 180,E1 -23993.753,E2 -23993.753} C_VEL
LIN {X 0,Y 170.967,Z 235.683,A -85,B 0,C 180,E1 -23994.944,E2 -23994.944} C_VEL
LIN {X 0,Y 170.005,Z 245.512,A -85,B 0,C 180,E1 -23995.631,E2 -23995.631} C_VEL
LIN {X 0,Y 168.371,Z 256.245,A -85,B 0,C 180,E1 -23996.737,E2 -23996.737} C_VEL
LIN {X 0,Y 166.028,Z 267.275,A -85,B 0,C 180,E1 -23998.409,E2 -23998.409} C_VEL
LIN {X 0,Y 163.814,Z 275.649,A -85,B 0,C 180,E1 -24000.083,E2 -24000.083} C_VEL
LIN {X 0,Y 161.293,Z 283.56,A -85,B 0,C 180,E1 -24002.068,E2 -24002.068} C_VEL
LIN {X 0,Y 158.707,Z 290.936,A -85,B 0,C 180,E1 -24004.42,E2 -24004.42} C_VEL
LIN {X 0,Y 155.874,Z 298.408,A -85,B 0,C 180,E1 -24007.465,E2 -24007.465} C_VEL
LIN {X 0,Y 152.971,Z 305.253,A -85,B 0,C 180,E1 -24011.239,E2 -24011.239} C_VEL
LIN {X 0,Y 150.787,Z 310.426,A -85,B 0,C 180,E1 -24015.146,E2 -24015.146} C_VEL
LIN {X 0,Y 149.634,Z 313.079,A -85,B 0,C 180,E1 -24017.798,E2 -24017.798} C_VEL
LIN {X 0,Y 148.479,Z 315.982,A -85,B 0,C 180,E1 -24021.836,E2 -24021.836} C_VEL
LIN {X 0,Y 148.006,Z 317.246,A -85,B 0,C 180,E1 -24024.55,E2 -24024.55} C_VEL
LIN {X 0,Y 147.631,Z 318.202,A -85,B 0,C 180,E1 -24028.637,E2 -24028.637} C_VEL
LIN {X 0,Y 147.623,Z 318.239,A -85,B 0,C 180,E1 -24031.227,E2 -24031.227} C_VEL
LIN {X 0,Y 148.002,Z 317.312,A -85,B 0,C 180,E1 -24035.449,E2 -24035.449} C_VEL
LIN {X 0,Y 148.403,Z 316.094,A -85,B 0,C 180,E1 -24038.167,E2 -24038.167} C_VEL
LIN {X 0,Y 149.627,Z 313.235,A -85,B 0,C 180,E1 -24042.202,E2 -24042.202} C_VEL
LIN {X 0,Y 150.728,Z 310.632,A -85,B 0,C 180,E1 -24044.859,E2 -24044.859} C_VEL
LIN {X 0,Y 152.935,Z 305.514,A -85,B 0,C 180,E1 -24048.764,E2 -24048.764} C_VEL
LIN {X 0,Y 155.298,Z 300.004,A -85,B 0,C 180,E1 -24051.922,E2 -24051.922} C_VEL
LIN {X 0,Y 158.028,Z 293.077,A -85,B 0,C 180,E1 -24054.991,E2 -24054.991} C_VEL
LIN {X 0,Y 160.909,Z 285.121,A -85,B 0,C 180,E1 -24057.649,E2 -24057.649} C_VEL
LIN {X 0,Y 163.415,Z 277.534,A -85,B 0,C 180,E1 -24059.641,E2 -24059.641} C_VEL
LIN {X 0,Y 165.581,Z 269.579,A -85,B 0,C 180,E1 -24061.328,E2 -24061.328} C_VEL
LIN {X 0,Y 167.54,Z 261.352,A -85,B 0,C 180,E1 -24062.689,E2 -24062.689} C_VEL
LIN {X 0,Y 169.076,Z 253.09,A -85,B 0,C 180,E1 -24063.763,E2 -24063.763} C_VEL
LIN {X 0,Y 170.436,Z 243.417,A -85,B 0,C 180,E1 -24064.686,E2 -24064.686} C_VEL
LIN {X 0,Y 171.315,Z 233.226,A -85,B 0,C 180,E1 -24065.335,E2 -24065.335} C_VEL
LIN {X 0,Y 172.711,Z 206.372,A -85,B 0,C 180,E1 -24066.393,E2 -24066.393} C_VEL
LIN {X 0,Y 168.309,Z 195.055,A -85,B 0,C 180,E1 -24068.109,E2 -24068.109} C_VEL
LIN {X 0,Y 164.891,Z 188.394,A -85,B 0,C 180,E1 -24069.418,E2 -24069.418} C_VEL
LIN {X 0,Y 160.319,Z 180.692,A -85,B 0,C 180,E1 -24071.228,E2 -24071.228} C_VEL
LIN {X 0,Y 155.465,Z 173.211,A -85,B 0,C 180,E1 -24073.285,E2 -24073.285} C_VEL
LIN {X 0,Y 153.334,Z 169.856,A -85,B 0,C 180,E1 -24074.258,E2 -24074.258} C_VEL
LIN {X 0,Y 150.932,Z 167.085,A -85,B 0,C 180,E1 -24075.34,E2 -24075.34} C_VEL
LIN {X 0,Y 150.269,Z 165.272,A -85,B 0,C 180,E1 -24075.872,E2 -24075.872} C_VEL
LIN {X 0,Y 150.131,Z 164.638,A -85,B 0,C 180,E1 -24076.66,E2 -24076.66} C_VEL
LIN {X 0,Y 150.172,Z 164.59,A -85,B 0,C 180,E1 -24082.526,E2 -24082.526} C_VEL
LIN {X 0,Y 150.219,Z 164.565,A -85,B 0,C 180,E1 -24087.364,E2 -24087.364} C_VEL
LIN {X 0,Y 150.244,Z 164.555,A -85,B 0,C 180,E1 -24092.717,E2 -24092.717} C_VEL
LIN {X 0,Y 150.35,Z 164.554,A -85,B 0,C 180,E1 -24099.207,E2 -24099.207} C_VEL
LIN {X 0,Y 150.381,Z 164.54,A -85,B 0,C 180,E1 -24103.715,E2 -24103.715} C_VEL
LIN {X 0,Y 150.652,Z 164.503,A -85,B 0,C 180,E1 -24109.245,E2 -24109.245} C_VEL
LIN {X 0,Y 150.724,Z 164.486,A -85,B 0,C 180,E1 -24111.959,E2 -24111.959} C_VEL
LIN {X 0,Y 151.218,Z 164.423,A -85,B 0,C 180,E1 -24120,E2 -24120} C_VEL
LIN {X 0,Y 150.745,Z 164.499,A -85,B 0,C 180,E1 -24128.04,E2 -24128.04} C_VEL
LIN {X 0,Y 150.607,Z 164.502,A -85,B 0,C 180,E1 -24131.496,E2 -24131.496} C_VEL
LIN {X 0,Y 150.382,Z 164.559,A -85,B 0,C 180,E1 -24136.284,E2 -24136.284} C_VEL
LIN {X 0,Y 150.35,Z 164.54,A -85,B 0,C 180,E1 -24140.792,E2 -24140.792} C_VEL
LIN {X 0,Y 150.243,Z 164.555,A -85,B 0,C 180,E1 -24147.282,E2 -24147.282} C_VEL
LIN {X 0,Y 150.218,Z 164.576,A -85,B 0,C 180,E1 -24152.635,E2 -24152.635} C_VEL
LIN {X 0,Y 150.176,Z 164.59,A -85,B 0,C 180,E1 -24157.472,E2 -24157.472} C_VEL
LIN {X 0,Y 150.126,Z 164.565,A -85,B 0,C 180,E1 -24162.921,E2 -24162.921} C_VEL
LIN {X 0,Y 150.217,Z 165.1,A -85,B 0,C 180,E1 -24163.829,E2 -24163.829} C_VEL
LIN {X 0,Y 151.26,Z 167.598,A -85,B 0,C 180,E1 -24164.61,E2 -24164.61} C_VEL
LIN {X 0,Y 153.352,Z 170.011,A -85,B 0,C 180,E1 -24165.55,E2 -24165.55} C_VEL
LIN {X 0,Y 155.559,Z 173.383,A -85,B 0,C 180,E1 -24166.549,E2 -24166.549} C_VEL
LIN {X 0,Y 159.793,Z 180.587,A -85,B 0,C 180,E1 -24168.39,E2 -24168.39} C_VEL
LIN {X 0,Y 165.109,Z 191.549,A -85,B 0,C 180,E1 -24170.609,E2 -24170.609} C_VEL
LIN {X 0,Y 170.065,Z 203.426,A -85,B 0,C 180,E1 -24172.582,E2 -24172.582} C_VEL
LIN {X 0,Y 171.135,Z 206.733,A -85,B 0,C 180,E1 -24173.025,E2 -24173.025} C_VEL
LIN {X 0,Y 172.195,Z 217.604,A -85,B 0,C 180,E1 -24173.84,E2 -24173.84} C_VEL
LIN {X 0,Y 170.837,Z 241.716,A -85,B 0,C 180,E1 -24174.835,E2 -24174.835} C_VEL
LIN {X 0,Y 169.464,Z 253.336,A -85,B 0,C 180,E1 -24175.667,E2 -24175.667} C_VEL
LIN {X 0,Y 167.427,Z 264.333,A -85,B 0,C 180,E1 -24176.929,E2 -24176.929} C_VEL
LIN {X 0,Y 165.478,Z 272.652,A -85,B 0,C 180,E1 -24178.212,E2 -24178.212} C_VEL
LIN {X 0,Y 163.143,Z 281.273,A -85,B 0,C 180,E1 -24179.949,E2 -24179.949} C_VEL
LIN {X 0,Y 160.585,Z 289.113,A -85,B 0,C 180,E1 -24181.936,E2 -24181.936} C_VEL
LIN {X 0,Y 157.996,Z 296.448,A -85,B 0,C 180,E1 -24184.298,E2 -24184.298} C_VEL
LIN {X 0,Y 155.114,Z 303.889,A -85,B 0,C 180,E1 -24187.349,E2 -24187.349} C_VEL
LIN {X 0,Y 152.251,Z 310.679,A -85,B 0,C 180,E1 -24191.149,E2 -24191.149} C_VEL
LIN {X 0,Y 150.138,Z 315.844,A -85,B 0,C 180,E1 -24195.082,E2 -24195.082} C_VEL
LIN {X 0,Y 148.713,Z 319.637,A -85,B 0,C 180,E1 -24199.104,E2 -24199.104} C_VEL
LIN {X 0,Y 148.049,Z 321.376,A -85,B 0,C 180,E1 -24201.813,E2 -24201.813} C_VEL
LIN {X 0,Y 147.704,Z 322.622,A -85,B 0,C 180,E1 -24204.54,E2 -24204.54} C_VEL
LIN {X 0,Y 147.57,Z 323.395,A -85,B 0,C 180,E1 -24207.271,E2 -24207.271} C_VEL
LIN {X 0,Y 147.596,Z 323.635,A -85,B 0,C 180,E1 -24210.614,E2 -24210.614} C_VEL
LIN {X 0,Y 147.57,Z 323.383,A -85,B 0,C 180,E1 -24212.73,E2 -24212.73} C_VEL
LIN {X 0,Y 147.703,Z 322.588,A -85,B 0,C 180,E1 -24215.461,E2 -24215.461} C_VEL
LIN {X 0,Y 148.041,Z 321.318,A -85,B 0,C 180,E1 -24218.189,E2 -24218.189} C_VEL
LIN {X 0,Y 149.066,Z 318.398,A -85,B 0,C 180,E1 -24222.25,E2 -24222.25} C_VEL
LIN {X 0,Y 149.208,Z 318.028,A -85,B 0,C 180,E1 -24222.673,E2 -24222.673} C_VEL
LIN {X 0,Y 149.366,Z 316.004,A -85,B 0,C 180,E1 -24224.804,E2 -24224.804} C_VEL
LIN {X 0,Y 148.222,Z 312.039,A -85,B 0,C 180,E1 -24228.283,E2 -24228.283} C_VEL
LIN {X 0,Y 147.545,Z 307.261,A -85,B 0,C 180,E1 -24231.643,E2 -24231.643} C_VEL
LIN {X 0,Y 148.407,Z 303.949,A -85,B 0,C 180,E1 -24233.51,E2 -24233.51} C_VEL
LIN {X 0,Y 151.643,Z 296.08,A -85,B 0,C 180,E1 -24236.864,E2 -24236.864} C_VEL
LIN {X 0,Y 154.34,Z 288.7,A -85,B 0,C 180,E1 -24239.309,E2 -24239.309} C_VEL
LIN {X 0,Y 157.023,Z 280.796,A -85,B 0,C 180,E1 -24241.354,E2 -24241.354} C_VEL
LIN {X 0,Y 159.87,Z 270.837,A -85,B 0,C 180,E1 -24243.358,E2 -24243.358} C_VEL
LIN {X 0,Y 162.262,Z 259.924,A -85,B 0,C 180,E1 -24244.937,E2 -24244.937} C_VEL
LIN {X 0,Y 163.994,Z 249.928,A -85,B 0,C 180,E1 -24245.925,E2 -24245.925} C_VEL
LIN {X 0,Y 165,Z 241.275,A -85,B 0,C 180,E1 -24246.521,E2 -24246.521} C_VEL
LIN {X 0,Y 166.331,Z 217.025,A -85,B 0,C 180,E1 -24247.566,E2 -24247.566} C_VEL
LIN {X 0,Y 165.228,Z 207.968,A -85,B 0,C 180,E1 -24248.348,E2 -24248.348} C_VEL
LIN {X 0,Y 161.514,Z 198.507,A -85,B 0,C 180,E1 -24249.926,E2 -24249.926} C_VEL
LIN {X 0,Y 156.374,Z 187.184,A -85,B 0,C 180,E1 -24252.195,E2 -24252.195} C_VEL
LIN {X 0,Y 151.992,Z 178.984,A -85,B 0,C 180,E1 -24254.229,E2 -24254.229} C_VEL
LIN {X 0,Y 149.508,Z 175.371,A -85,B 0,C 180,E1 -24255.399,E2 -24255.399} C_VEL
LIN {X 0,Y 146.782,Z 171.646,A -85,B 0,C 180,E1 -24256.742,E2 -24256.742} C_VEL
LIN {X 0,Y 145.959,Z 170.287,A -85,B 0,C 180,E1 -24257.181,E2 -24257.181} C_VEL
LIN {X 0,Y 143.995,Z 168.12,A -85,B 0,C 180,E1 -24258.184,E2 -24258.184} C_VEL
LIN {X 0,Y 143.204,Z 166.054,A -85,B 0,C 180,E1 -24258.894,E2 -24258.894} C_VEL
LIN {X 0,Y 143.065,Z 165.469,A -85,B 0,C 180,E1 -24259.988,E2 -24259.988} C_VEL
LIN {X 0,Y 143.09,Z 165.455,A -85,B 0,C 180,E1 -24263.886,E2 -24263.886} C_VEL
LIN {X 0,Y 143.188,Z 165.451,A -85,B 0,C 180,E1 -24267.323,E2 -24267.323} C_VEL
LIN {X 0,Y 143.193,Z 165.432,A -85,B 0,C 180,E1 -24272.062,E2 -24272.062} C_VEL
LIN {X 0,Y 143.279,Z 165.423,A -85,B 0,C 180,E1 -24278.746,E2 -24278.746} C_VEL
LIN {X 0,Y 143.315,Z 165.428,A -85,B 0,C 180,E1 -24282.889,E2 -24282.889} C_VEL
LIN {X 0,Y 143.54,Z 165.38,A -85,B 0,C 180,E1 -24288.706,E2 -24288.706} C_VEL
LIN {X 0,Y 143.63,Z 165.378,A -85,B 0,C 180,E1 -24291.559,E2 -24291.559} C_VEL
LIN {X 0,Y 144.178,Z 165.298,A -85,B 0,C 180,E1 -24300,E2 -24300} C_VEL
LIN {X 0,Y 143.651,Z 165.364,A -85,B 0,C 180,E1 -24308.44,E2 -24308.44} C_VEL
LIN {X 0,Y 143.55,Z 165.397,A -85,B 0,C 180,E1 -24311.713,E2 -24311.713} C_VEL
LIN {X 0,Y 143.318,Z 165.412,A -85,B 0,C 180,E1 -24317.111,E2 -24317.111} C_VEL
LIN {X 0,Y 143.283,Z 165.437,A -85,B 0,C 180,E1 -24321.259,E2 -24321.259} C_VEL
LIN {X 0,Y 143.194,Z 165.435,A -85,B 0,C 180,E1 -24327.938,E2 -24327.938} C_VEL
LIN {X 0,Y 143.149,Z 165.442,A -85,B 0,C 180,E1 -24333.422,E2 -24333.422} C_VEL
LIN {X 0,Y 143.063,Z 165.459,A -85,B 0,C 180,E1 -24339.69,E2 -24339.69} C_VEL
LIN {X 0,Y 143.155,Z 165.786,A -85,B 0,C 180,E1 -24341.212,E2 -24341.212} C_VEL
LIN {X 0,Y 143.459,Z 166.979,A -85,B 0,C 180,E1 -24341.767,E2 -24341.767} C_VEL
LIN {X 0,Y 145.09,Z 169.589,A -85,B 0,C 180,E1 -24342.699,E2 -24342.699} C_VEL
LIN {X 0,Y 146.461,Z 170.961,A -85,B 0,C 180,E1 -24343.377,E2 -24343.377} C_VEL
LIN {X 0,Y 148.46,Z 174.113,A -85,B 0,C 180,E1 -24344.406,E2 -24344.406} C_VEL
LIN {X 0,Y 149.848,Z 175.949,A -85,B 0,C 180,E1 -24345.07,E2 -24345.07} C_VEL
LIN {X 0,Y 156.453,Z 186.108,A -85,B 0,C 180,E1 -24348.066,E2 -24348.066} C_VEL
LIN {X 0,Y 162.639,Z 197.252,A -85,B 0,C 180,E1 -24350.632,E2 -24350.632} C_VEL
LIN {X 0,Y 166.829,Z 208.003,A -85,B 0,C 180,E1 -24352.385,E2 -24352.385} C_VEL
LIN {X 0,Y 165.169,Z 236.766,A -85,B 0,C 180,E1 -24353.589,E2 -24353.589} C_VEL
LIN {X 0,Y 163.944,Z 247.58,A -85,B 0,C 180,E1 -24354.389,E2 -24354.389} C_VEL
LIN {X 0,Y 162.05,Z 258.615,A -85,B 0,C 180,E1 -24355.68,E2 -24355.68} C_VEL
LIN {X 0,Y 160.037,Z 267.408,A -85,B 0,C 180,E1 -24357.081,E2 -24357.081} C_VEL
LIN {X 0,Y 157.703,Z 275.781,A -85,B 0,C 180,E1 -24358.797,E2 -24358.797} C_VEL
LIN {X 0,Y 155.075,Z 283.691,A -85,B 0,C 180,E1 -24360.843,E2 -24360.843} C_VEL
LIN {X 0,Y 152.348,Z 291.067,A -85,B 0,C 180,E1 -24363.27,E2 -24363.27} C_VEL
LIN {X 0,Y 149.343,Z 298.538,A -85,B 0,C 180,E1 -24366.421,E2 -24366.421} C_VEL
LIN {X 0,Y 146.272,Z 305.383,A -85,B 0,C 180,E1 -24370.346,E2 -24370.346} C_VEL
LIN {X 0,Y 143.925,Z 310.556,A -85,B 0,C 180,E1 -24374.42,E2 -24374.42} C_VEL
LIN {X 0,Y 142.712,Z 313.208,A -85,B 0,C 180,E1 -24377.196,E2 -24377.196} C_VEL
LIN {X 0,Y 141.446,Z 316.111,A -85,B 0,C 180,E1 -24381.427,E2 -24381.427} C_VEL
LIN {X 0,Y 140.945,Z 317.375,A -85,B 0,C 180,E1 -24384.276,E2 -24384.276} C_VEL
LIN {X 0,Y 140.623,Z 318.171,A -85,B 0,C 180,E1 -24387.135,E2 -24387.135} C_VEL
LIN {X 0,Y 140.561,Z 318.473,A -85,B 0,C 180,E1 -24389.999,E2 -24389.999} C_VEL
LIN {X 0,Y 140.622,Z 318.192,A -85,B 0,C 180,E1 -24392.864,E2 -24392.864} C_VEL
LIN {X 0,Y 140.941,Z 317.44,A -85,B 0,C 180,E1 -24395.723,E2 -24395.723} C_VEL
LIN {X 0,Y 141.39,Z 316.221,A -85,B 0,C 180,E1 -24398.575,E2 -24398.575} C_VEL
LIN {X 0,Y 142.704,Z 313.362,A -85,B 0,C 180,E1 -24402.803,E2 -24402.803} C_VEL
LIN {X 0,Y 143.873,Z 310.76,A -85,B 0,C 180,E1 -24405.584,E2 -24405.584} C_VEL
LIN {X 0,Y 146.231,Z 305.641,A -85,B 0,C 180,E1 -24409.659,E2 -24409.659} C_VEL
LIN {X 0,Y 148.739,Z 300.131,A -85,B 0,C 180,E1 -24412.942,E2 -24412.942} C_VEL
LIN {X 0,Y 151.616,Z 293.203,A -85,B 0,C 180,E1 -24416.126,E2 -24416.126} C_VEL
LIN {X 0,Y 154.662,Z 285.246,A -85,B 0,C 180,E1 -24418.868,E2 -24418.868} C_VEL
LIN {X 0,Y 157.295,Z 277.658,A -85,B 0,C 180,E1 -24420.918,E2 -24420.918} C_VEL
LIN {X 0,Y 159.562,Z 269.702,A -85,B 0,C 180,E1 -24422.653,E2 -24422.653} C_VEL
LIN {X 0,Y 161.624,Z 261.474,A -85,B 0,C 180,E1 -24424.045,E2 -24424.045} C_VEL
LIN {X 0,Y 163.252,Z 253.074,A -85,B 0,C 180,E1 -24425.162,E2 -24425.162} C_VEL
LIN {X 0,Y 164.639,Z 243.734,A -85,B 0,C 180,E1 -24426.072,E2 -24426.072} C_VEL
LIN {X 0,Y 165.535,Z 234.028,A -85,B 0,C 180,E1 -24426.716,E2 -24426.716} C_VEL
LIN {X 0,Y 166.982,Z 208.122,A -85,B 0,C 180,E1 -24427.768,E2 -24427.768} C_VEL
LIN {X 0,Y 162.272,Z 196.425,A -85,B 0,C 180,E1 -24429.73,E2 -24429.73} C_VEL
LIN {X 0,Y 156.349,Z 185.895,A -85,B 0,C 180,E1 -24432.203,E2 -24432.203} C_VEL
LIN {X 0,Y 151.074,Z 177.812,A -85,B 0,C 180,E1 -24434.579,E2 -24434.579} C_VEL
LIN {X 0,Y 149.027,Z 174.716,A -85,B 0,C 180,E1 -24435.571,E2 -24435.571} C_VEL
LIN {X 0,Y 146.857,Z 171.758,A -85,B 0,C 180,E1 -24436.651,E2 -24436.651} C_VEL
LIN {X 0,Y 145.91,Z 170.276,A -85,B 0,C 180,E1 -24437.153,E2 -24437.153} C_VEL
LIN {X 0,Y 143.958,Z 168.081,A -85,B 0,C 180,E1 -24438.161,E2 -24438.161} C_VEL
LIN {X 0,Y 143.214,Z 165.987,A -85,B 0,C 180,E1 -24438.892,E2 -24438.892} C_VEL
LIN {X 0,Y 143.087,Z 165.514,A -85,B 0,C 180,E1 -24439.668,E2 -24439.668} C_VEL
LIN {X 0,Y 143.087,Z 165.465,A -85,B 0,C 180,E1 -24443.885,E2 -24443.885} C_VEL
LIN {X 0,Y 143.186,Z 165.44,A -85,B 0,C 180,E1 -24447.322,E2 -24447.322} C_VEL
LIN {X 0,Y 143.192,Z 165.436,A -85,B 0,C 180,E1 -24452.061,E2 -24452.061} C_VEL
LIN {X 0,Y 143.28,Z 165.44,A -85,B 0,C 180,E1 -24458.741,E2 -24458.741} C_VEL
LIN {X 0,Y 143.315,Z 165.412,A -85,B 0,C 180,E1 -24462.888,E2 -24462.888} C_VEL
LIN {X 0,Y 143.593,Z 165.386,A -85,B 0,C 180,E1 -24468.71,E2 -24468.71} C_VEL
LIN {X 0,Y 143.648,Z 165.365,A -85,B 0,C 180,E1 -24471.56,E2 -24471.56} C_VEL
LIN {X 0,Y 144.176,Z 165.299,A -85,B 0,C 180,E1 -24480,E2 -24480} C_VEL
LIN {X 0,Y 143.664,Z 165.374,A -85,B 0,C 180,E1 -24488.439,E2 -24488.439} C_VEL
LIN {X 0,Y 143.547,Z 165.382,A -85,B 0,C 180,E1 -24491.712,E2 -24491.712} C_VEL
LIN {X 0,Y 143.316,Z 165.427,A -85,B 0,C 180,E1 -24497.111,E2 -24497.111} C_VEL
LIN {X 0,Y 143.275,Z 165.424,A -85,B 0,C 180,E1 -24501.254,E2 -24501.254} C_VEL
LIN {X 0,Y 143.19,Z 165.432,A -85,B 0,C 180,E1 -24507.938,E2 -24507.938} C_VEL
LIN {X 0,Y 143.146,Z 165.448,A -85,B 0,C 180,E1 -24513.422,E2 -24513.422} C_VEL
LIN {X 0,Y 143.054,Z 165.45,A -85,B 0,C 180,E1 -24519.692,E2 -24519.692} C_VEL
LIN {X 0,Y 143.161,Z 165.842,A -85,B 0,C 180,E1 -24520.793,E2 -24520.793} C_VEL
LIN {X 0,Y 143.582,Z 167.236,A -85,B 0,C 180,E1 -24521.384,E2 -24521.384} C_VEL
